(* CoDeSys 2.3.9.41 project: GermesLib_1_2.pro *)
(* Libraries: PID_Regulators.lib 6.11.19 15:29:27, Util.lib 18.5.10 15:14:28, STANDARD.LIB 4.10.05 11:14:46, IECSFC.LIB 13.4.06 15:51:28, ANALYZATION.LIB 5.10.99 09:05:06 *)

(* PLC configuration (modules and I/O channels)
Fast discrete inputs [I_SIMPLE_INPUT] node 0, in %IB0 out %QB0 {Filtrationtime = 10}
  DD1_DI0 AT %IX0.0 [BitInput] резерв
  DD1_DI1 AT %IX0.1 [BitInput] резерв
  DD1_DI2 AT %IX0.2 [BitInput] резерв
  DD1_DI3 AT %IX0.3 [BitInput] резерв
Discrete inputs [ID130] node 1, in %IB1 out %QB1 {Filtrationtime_GeneralINP = 10; Visibility = No; PinCount = 12}
  AT %IB1.0 [ByteInput] 8 discrete inputs
  AT %IB1.1 [ByteInput] 4 discrete inputs
Discrete outputs [ID131] node 2, in %IB2 out %QB2 {SafeValueByte = 0; SafeValueByteM = 0; Visibility = No; PinCount = 12}
  AT %QB2.0 [ByteOutput] 8 discrete outputs
  AT %QB2.1 [ByteOutput] 4 discrete outputs
Fast analog inputs [ID125] node 3, in %IB3 out %QB3 {Flt_Comm = 50Hz 2Por}
  DD1_AI0 AT %IR3.0 [FloatInputP] AI #1 - датчик температуры в помещении (метран) {AIN_TYPE = 4-20 mA; Peak_Filtr = 200; Flt_Ch = Off; TauRC = 10; MinFV = 0; MaxFV = 100}
  DD1_AI1 AT %IR3.1 [FloatInputP] AI #2 - расходомер FT01.01 (на входе, до отстойника) {AIN_TYPE = 4-20 mA; Peak_Filtr = 200; Flt_Ch = Off; TauRC = 10; MinFV = 0; MaxFV = 600}
  DD1_AI2 AT %IR3.2 [FloatInputP] AI #3 - расходомер FT01.02 (на выходе, после отстойника) {AIN_TYPE = 4-20 mA; Peak_Filtr = 200; Flt_Ch = Off; TauRC = 10; MinFV = 0; MaxFV = 600}
  DD1_AI3 AT %IR3.3 [FloatInputP] AI #4 - рН-метр QE01.01 (на входе, до отстойника) {AIN_TYPE = 4-20 mA; Peak_Filtr = 200; Flt_Ch = Off; TauRC = 10; MinFV = 0; MaxFV = 14}
  DD1_AI4 AT %IR3.4 [FloatInputP] AI #5 - рН-метр QE01.02 (на выходе, после отстойника) {AIN_TYPE = 4-20 mA; Peak_Filtr = 200; Flt_Ch = Off; TauRC = 10; MinFV = 0; MaxFV = 14}
  DD1_AI5 AT %IR3.5 [FloatInputP] AI #6 - сигнал от ФПК, давление на входе {AIN_TYPE = 4-20 mA; Peak_Filtr = 200; Flt_Ch = Off; TauRC = 10; MinFV = 0; MaxFV = 16}
  DD1_AI6 AT %IR3.6 [FloatInputP] AI #7 - резерв {AIN_TYPE = 4-20 mA; Peak_Filtr = 200; Flt_Ch = Off; TauRC = 10; MinFV = 0; MaxFV = 20000.0}
  DD1_AI7 AT %IR3.7 [FloatInputP] AI#8 - резерв {AIN_TYPE = 4-20 mA; Peak_Filtr = 200; Flt_Ch = Off; TauRC = 10; MinFV = 0; MaxFV = 20000.0}
  AT %IW3.8 [WordInput] AI read time (10ms)
Analog outputs [ID126] node 4, in %IB4 out %QB4
  DD1_AO0 AT %QR4.0 [FloatOutputP] AO #1 - управление ЧРП Н01.05 (поддержание расхода по расходомеру FT01.02) {AOUT_TYPE = 4-20 mA; SafeValueREAL = 0.0}
  DD1_AO1 AT %QR4.1 [FloatOutputP] AO #2 - управление ЧРП НД08.03/01 (подача флокулянта на входе, до отстойника, по FT01.01) {AOUT_TYPE = 4-20 mA; SafeValueREAL = 0.0}
  DD1_AO2 AT %QR4.2 [FloatOutputP] AO #3 - управление ЧРП НД08.03/02 (подача флокулянта на входе, до отстойника, по FT01.01) {AOUT_TYPE = 4-20 mA; SafeValueREAL = 0.0}
  DD1_AO3 AT %QR4.3 [FloatOutputP] AO #4 - управление НД05.02/01 (подача 10%NaCl из УПГ на входе, до отстойника, по FT01.01) {AOUT_TYPE = 4-20 mA; SafeValueREAL = 0.0}
Special input [ID103] node 5, in %IB5 out %QB5 {Filtrationtime = 1000; PinCount = 1; WatchDogPeriod = 400; PollPeriod = 3000; Visibility = No}
  AT %IX5.0 [BitInput] Special input
Special output [ID104] node 6, in %IB6 out %QB6 {Visibility = No; PinCount = 1}
  AT %QX6.0 [BitOutput] Special output
lastAddress AT %QD7.0 [DWordOutput] Last address
lastError AT %QW7.1 [WordOutput] Last error
RS-485-1 [COM1_USART] node 0, in %IB7.0 out %QB7.0 {CommunicationSpeed = 9600; Parity = EVEN; BitLength = 8 bits; StopLength = One stop bit; InterfaceType = RS485; FrameOriented = RTU; Timeout = 0; Visibility = No}
Universal Modbus device [ID2000] node 1, in %IB7.1 out %QB7.1 {ModuleIP = 10:0:0:102; ServiceTimeout = 20; TCPport = 502; NetMode = Serial; ModuleSlaveAddress = 2; RequestType = Both; PeriodOfService = 100; Visibility = No; RepeatCounter = 0; ByteSequence = Trace_mode}
  AT %QB7.1.0 [ComChannel] Command (0xff - Start)
DD2_DO AT %QD7.1.0.0 [DWordOutput] регистр 0, команда 0х0f
Universal Modbus device [ID2000] node 2, in %IB7.2 out %QB7.2 {ModuleIP = 10:0:0:103; ServiceTimeout = 20; TCPport = 502; NetMode = Serial; ModuleSlaveAddress = 3; RequestType = Both; PeriodOfService = 100; Visibility = No; RepeatCounter = 0; ByteSequence = Trace_mode}
  AT %QB7.2.0 [ComChannel] Command (0xff - Start)
DD3_DO AT %QD7.2.0.0 [DWordOutput]
Universal Modbus device [ID2000] node 3, in %IB7.3 out %QB7.3 {ModuleIP = 10:0:0:104; ServiceTimeout = 20; TCPport = 502; NetMode = Serial; ModuleSlaveAddress = 4; RequestType = Both; PeriodOfService = 100; Visibility = No; RepeatCounter = 0; ByteSequence = Trace_mode}
  AT %QB7.3.0 [ComChannel] Command (0xff - Start)
  32bit output module [ID2006] node 0, in %IB7.3.0 out %QB7.3.0 {ModbusAddress = 0; Command_write_regs = Force multiple coils (0x0f); Visibility = No}
    DD4_DO AT %QD7.3.0.0 [DWordOutput]
Universal Modbus device [ID2000] node 4, in %IB7.4 out %QB7.4 {ModuleIP = 10:0:0:105; ServiceTimeout = 20; TCPport = 502; NetMode = Serial; ModuleSlaveAddress = 5; RequestType = Both; PeriodOfService = 100; Visibility = No; RepeatCounter = 0; ByteSequence = Trace_mode}
  AT %QB7.4.0 [ComChannel] Command (0xff - Start)
DD5_DI AT %ID7.4.0.0 [DWordInput]
Universal Modbus device [ID2000] node 5, in %IB7.5 out %QB7.5 {ModuleIP = 10:0:0:106; ServiceTimeout = 20; TCPport = 502; NetMode = Serial; ModuleSlaveAddress = 6; RequestType = Both; PeriodOfService = 100; Visibility = No; RepeatCounter = 0; ByteSequence = Trace_mode}
  AT %QB7.5.0 [ComChannel] Command (0xff - Start)
DD6_DI AT %ID7.5.0.0 [DWordInput]
Universal Modbus device [ID2000] node 6, in %IB7.6 out %QB7.6 {ModuleIP = 10:0:0:107; ServiceTimeout = 20; TCPport = 502; NetMode = Serial; ModuleSlaveAddress = 7; RequestType = Both; PeriodOfService = 100; Visibility = No; RepeatCounter = 0; ByteSequence = Trace_mode}
  AT %QB7.6.0 [ComChannel] Command (0xff - Start)
DD7_DI AT %ID7.6.0.0 [DWordInput]
Universal Modbus device [ID2000] node 7, in %IB7.7 out %QB7.7 {ModuleIP = 10:0:0:108; ServiceTimeout = 20; TCPport = 502; NetMode = Serial; ModuleSlaveAddress = 8; RequestType = Both; PeriodOfService = 100; Visibility = No; RepeatCounter = 0; ByteSequence = Trace_mode}
  AT %QB7.7.0 [ComChannel] Command (0xff - Start)
DD8_DI AT %ID7.7.0.0 [DWordInput]
Universal Modbus device [ID2000] node 8, in %IB7.8 out %QB7.8 {ModuleIP = 10:0:0:109; ServiceTimeout = 20; TCPport = 502; NetMode = Serial; ModuleSlaveAddress = 9; RequestType = Both; PeriodOfService = 100; Visibility = No; RepeatCounter = 0; ByteSequence = Trace_mode}
  AT %QB7.8.0 [ComChannel] Command (0xff - Start)
DD9_DI AT %ID7.8.0.0 [DWordInput]
Universal Modbus device [ID2000] node 9, in %IB7.9 out %QB7.9 {ModuleIP = 10:0:0:110; ServiceTimeout = 20; TCPport = 502; NetMode = Serial; ModuleSlaveAddress = 10; RequestType = Both; PeriodOfService = 100; Visibility = No; RepeatCounter = 0; ByteSequence = Trace_mode}
  AT %QB7.9.0 [ComChannel] Command (0xff - Start)
DD10_AO0 AT %QW7.9.0.0 [WordOutput] управление 4...20мА НД05.02/02
DD10_AO1 AT %QW7.9.1.0 [WordOutput] управление 4...20мА НД06.02/01
DD10_AO2 AT %QW7.9.2.0 [WordOutput] управление 4...20мА НД06.02/02
DD10_AO3 AT %QW7.9.3.0 [WordOutput] управление 4...20мА НД06.03/01
DD10_AO4 AT %QW7.9.4.0 [WordOutput] управление 4...20мА НД06.03/02
DD10_AO5 AT %QW7.9.5.0 [WordOutput] управление 4...20мА НД07.03/01
DD10_AO6 AT %QW7.9.6.0 [WordOutput] управление 4...20мА НД07.03/02
DD10_AO7 AT %QW7.9.7.0 [WordOutput] управление 4...20мА НД08.04
Universal Modbus device [ID2000] node 10, in %IB7.10 out %QB7.10 {ModuleIP = 10:0:0:223; ServiceTimeout = 20; TCPport = 502; NetMode = Serial; ModuleSlaveAddress = 11; RequestType = By value change; PeriodOfService = 100; Visibility = No; RepeatCounter = 0; ByteSequence = Trace_mode}
  AT %QB7.10.0 [ComChannel] Command (0xff - Start)
AT %QB7.10.0.0 [ByteOutput]
Universal Modbus device [ID2000] node 11, in %IB7.11 out %QB7.11 {ModuleIP = 10:0:0:223; ServiceTimeout = 20; TCPport = 502; NetMode = Serial; ModuleSlaveAddress = 11; RequestType = By poll time; PeriodOfService = 100; Visibility = No; RepeatCounter = 0; ByteSequence = Trace_mode}
  AT %QB7.11.0 [ComChannel] Command (0xff - Start)
AT %IB7.11.0.0 [ByteInput]
Universal Modbus device [ID2000] node 12, in %IB7.12 out %QB7.12 {ModuleIP = 10:0:0:223; ServiceTimeout = 20; TCPport = 502; NetMode = Serial; ModuleSlaveAddress = 12; RequestType = By value change; PeriodOfService = 100; Visibility = No; RepeatCounter = 0; ByteSequence = Trace_mode}
  AT %QB7.12.0 [ComChannel] Command (0xff - Start)
AT %QB7.12.0.0 [ByteOutput]
Universal Modbus device [ID2000] node 13, in %IB7.13 out %QB7.13 {ModuleIP = 10:0:0:223; ServiceTimeout = 20; TCPport = 502; NetMode = Serial; ModuleSlaveAddress = 12; RequestType = By poll time; PeriodOfService = 100; Visibility = No; RepeatCounter = 0; ByteSequence = Trace_mode}
  AT %QB7.13.0 [ComChannel] Command (0xff - Start)
AT %IB7.13.0.0 [ByteInput]
AT %QD8.0 [DWordOutput] Last address
AT %QW8.1 [WordOutput] Last error
RS-232 [COM2_USART] node 0, in %IB8.0 out %QB8.0 {CommunicationSpeed = 57600; Parity = NO PARITY CHECK; BitLength = 8 bits; StopLength = One stop bit; InterfaceType = RS232; FrameOriented = RTU; Timeout = 0; Visibility = No}
AT %QB8.1.0 [ComChannel] Command (0xff - Start)
Real output module [ID2008] node 0, in %IB8.1.0 out %QB8.1.0 {ModbusAddress = 256; Command_write_regs = Preset multiple Registers (0x10); Visibility = No}
  panFT0101value AT %QD8.1.0.0 [FloatOutput]
Real output module [ID2008] node 1, in %IB8.1.1 out %QB8.1.1 {ModbusAddress = 258; Command_write_regs = Preset multiple Registers (0x10); Visibility = No}
  panQE0101value AT %QD8.1.1.0 [FloatOutput]
Real output module [ID2008] node 2, in %IB8.1.2 out %QB8.1.2 {ModbusAddress = 260; Command_write_regs = Preset multiple Registers (0x10); Visibility = No}
  panFT0102value AT %QD8.1.2.0 [FloatOutput]
Real output module [ID2008] node 3, in %IB8.1.3 out %QB8.1.3 {ModbusAddress = 262; Command_write_regs = Preset multiple Registers (0x10); Visibility = No}
  panQE0102value AT %QD8.1.3.0 [FloatOutput]
Real output module [ID2008] node 4, in %IB8.1.4 out %QB8.1.4 {ModbusAddress = 264; Command_write_regs = Preset multiple Registers (0x10); Visibility = No}
  panFPKpressureValue AT %QD8.1.4.0 [FloatOutput]
Real output module [ID2008] node 5, in %IB8.1.5 out %QB8.1.5 {ModbusAddress = 266; Command_write_regs = Preset multiple Registers (0x10); Visibility = No}
  panFQS0301total AT %QD8.1.5.0 [FloatOutput]
Real output module [ID2008] node 6, in %IB8.1.6 out %QB8.1.6 {ModbusAddress = 268; Command_write_regs = Preset multiple Registers (0x10); Visibility = No}
  panTemperature AT %QD8.1.6.0 [FloatOutput]
Register output module [ID2004] node 7, in %IB8.1.7 out %QB8.1.7 {ModbusAddress = 270; Command_write_one_reg = Write multiple registers(0x10); Visibility = No}
  panND050201workDays AT %QW8.1.7.0 [WordOutput]
Register output module [ID2004] node 8, in %IB8.1.8 out %QB8.1.8 {ModbusAddress = 271; Command_write_one_reg = Write multiple registers(0x10); Visibility = No}
  panND050201workHours AT %QW8.1.8.0 [WordOutput]
Register output module [ID2004] node 9, in %IB8.1.9 out %QB8.1.9 {ModbusAddress = 272; Command_write_one_reg = Write multiple registers(0x10); Visibility = No}
  panND050201workMinutes AT %QW8.1.9.0 [WordOutput]
Register output module [ID2004] node 10, in %IB8.1.10 out %QB8.1.10 {ModbusAddress = 273; Command_write_one_reg = Write multiple registers(0x10); Visibility = No}
  panND050201workSeconds AT %QW8.1.10.0 [WordOutput]
Register output module [ID2004] node 11, in %IB8.1.11 out %QB8.1.11 {ModbusAddress = 274; Command_write_one_reg = Write multiple registers(0x10); Visibility = No}
  panND050202workDays AT %QW8.1.11.0 [WordOutput]
Register output module [ID2004] node 12, in %IB8.1.12 out %QB8.1.12 {ModbusAddress = 275; Command_write_one_reg = Write multiple registers(0x10); Visibility = No}
  panND050202workHours AT %QW8.1.12.0 [WordOutput]
Register output module [ID2004] node 13, in %IB8.1.13 out %QB8.1.13 {ModbusAddress = 276; Command_write_one_reg = Write multiple registers(0x10); Visibility = No}
  panND050202workMinutes AT %QW8.1.13.0 [WordOutput]
Register output module [ID2004] node 14, in %IB8.1.14 out %QB8.1.14 {ModbusAddress = 277; Command_write_one_reg = Write multiple registers(0x10); Visibility = No}
  panND050202workSeconds AT %QW8.1.14.0 [WordOutput]
Register output module [ID2004] node 15, in %IB8.1.15 out %QB8.1.15 {ModbusAddress = 278; Command_write_one_reg = Write multiple registers(0x10); Visibility = No}
  panND0502counterP1 AT %QW8.1.15.0 [WordOutput]
Register output module [ID2004] node 16, in %IB8.1.16 out %QB8.1.16 {ModbusAddress = 279; Command_write_one_reg = Write multiple registers(0x10); Visibility = No}
  panND0502counterP2 AT %QW8.1.16.0 [WordOutput]
Register output module [ID2004] node 17, in %IB8.1.17 out %QB8.1.17 {ModbusAddress = 280; Command_write_one_reg = Write multiple registers(0x10); Visibility = No}
  panND060201workDays AT %QW8.1.17.0 [WordOutput]
Register output module [ID2004] node 18, in %IB8.1.18 out %QB8.1.18 {ModbusAddress = 281; Command_write_one_reg = Write multiple registers(0x10); Visibility = No}
  panND060201workHours AT %QW8.1.18.0 [WordOutput]
Register output module [ID2004] node 19, in %IB8.1.19 out %QB8.1.19 {ModbusAddress = 282; Command_write_one_reg = Write multiple registers(0x10); Visibility = No}
  panND060201workMinutes AT %QW8.1.19.0 [WordOutput]
Register output module [ID2004] node 20, in %IB8.1.20 out %QB8.1.20 {ModbusAddress = 283; Command_write_one_reg = Write multiple registers(0x10); Visibility = No}
  panND060201workSeconds AT %QW8.1.20.0 [WordOutput]
Register output module [ID2004] node 21, in %IB8.1.21 out %QB8.1.21 {ModbusAddress = 284; Command_write_one_reg = Write multiple registers(0x10); Visibility = No}
  panND060202workDays AT %QW8.1.21.0 [WordOutput]
Register output module [ID2004] node 22, in %IB8.1.22 out %QB8.1.22 {ModbusAddress = 285; Command_write_one_reg = Write multiple registers(0x10); Visibility = No}
  panND060202workHours AT %QW8.1.22.0 [WordOutput]
Register output module [ID2004] node 23, in %IB8.1.23 out %QB8.1.23 {ModbusAddress = 286; Command_write_one_reg = Write multiple registers(0x10); Visibility = No}
  panND060202workMinutes AT %QW8.1.23.0 [WordOutput]
Register output module [ID2004] node 24, in %IB8.1.24 out %QB8.1.24 {ModbusAddress = 287; Command_write_one_reg = Write multiple registers(0x10); Visibility = No}
  panND060202workSeconds AT %QW8.1.24.0 [WordOutput]
Register output module [ID2004] node 25, in %IB8.1.25 out %QB8.1.25 {ModbusAddress = 288; Command_write_one_reg = Write multiple registers(0x10); Visibility = No}
  panND0602counterP1 AT %QW8.1.25.0 [WordOutput]
Register output module [ID2004] node 26, in %IB8.1.26 out %QB8.1.26 {ModbusAddress = 289; Command_write_one_reg = Write multiple registers(0x10); Visibility = No}
  panND0602counterP2 AT %QW8.1.26.0 [WordOutput]
Register output module [ID2004] node 27, in %IB8.1.27 out %QB8.1.27 {ModbusAddress = 290; Command_write_one_reg = Write multiple registers(0x10); Visibility = No}
  panND060301workDays AT %QW8.1.27.0 [WordOutput]
Register output module [ID2004] node 28, in %IB8.1.28 out %QB8.1.28 {ModbusAddress = 291; Command_write_one_reg = Write multiple registers(0x10); Visibility = No}
  panND060301workHours AT %QW8.1.28.0 [WordOutput]
Register output module [ID2004] node 29, in %IB8.1.29 out %QB8.1.29 {ModbusAddress = 292; Command_write_one_reg = Write multiple registers(0x10); Visibility = No}
  panND060301workMinutes AT %QW8.1.29.0 [WordOutput]
Register output module [ID2004] node 30, in %IB8.1.30 out %QB8.1.30 {ModbusAddress = 293; Command_write_one_reg = Write multiple registers(0x10); Visibility = No}
  panND060301workSeconds AT %QW8.1.30.0 [WordOutput]
Register output module [ID2004] node 31, in %IB8.1.31 out %QB8.1.31 {ModbusAddress = 294; Command_write_one_reg = Write multiple registers(0x10); Visibility = No}
  panND060302workDays AT %QW8.1.31.0 [WordOutput]
Register output module [ID2004] node 32, in %IB8.1.32 out %QB8.1.32 {ModbusAddress = 295; Command_write_one_reg = Write multiple registers(0x10); Visibility = No}
  panND060302workHours AT %QW8.1.32.0 [WordOutput]
Register output module [ID2004] node 33, in %IB8.1.33 out %QB8.1.33 {ModbusAddress = 296; Command_write_one_reg = Write multiple registers(0x10); Visibility = No}
  panND060302workMinutes AT %QW8.1.33.0 [WordOutput]
Register output module [ID2004] node 34, in %IB8.1.34 out %QB8.1.34 {ModbusAddress = 297; Command_write_one_reg = Write multiple registers(0x10); Visibility = No}
  panND060302workSeconds AT %QW8.1.34.0 [WordOutput]
Register output module [ID2004] node 35, in %IB8.1.35 out %QB8.1.35 {ModbusAddress = 298; Command_write_one_reg = Write multiple registers(0x10); Visibility = No}
  panND0603counterP1 AT %QW8.1.35.0 [WordOutput]
Register output module [ID2004] node 36, in %IB8.1.36 out %QB8.1.36 {ModbusAddress = 299; Command_write_one_reg = Write multiple registers(0x10); Visibility = No}
  panND0603counterP2 AT %QW8.1.36.0 [WordOutput]
Register output module [ID2004] node 37, in %IB8.1.37 out %QB8.1.37 {ModbusAddress = 300; Command_write_one_reg = Write multiple registers(0x10); Visibility = No}
  panND070301workDays AT %QW8.1.37.0 [WordOutput]
Register output module [ID2004] node 38, in %IB8.1.38 out %QB8.1.38 {ModbusAddress = 301; Command_write_one_reg = Write multiple registers(0x10); Visibility = No}
  panND070301workHours AT %QW8.1.38.0 [WordOutput]
Register output module [ID2004] node 39, in %IB8.1.39 out %QB8.1.39 {ModbusAddress = 302; Command_write_one_reg = Write multiple registers(0x10); Visibility = No}
  panND070301workMinutes AT %QW8.1.39.0 [WordOutput]
Register output module [ID2004] node 40, in %IB8.1.40 out %QB8.1.40 {ModbusAddress = 303; Command_write_one_reg = Write multiple registers(0x10); Visibility = No}
  panND070301workSeconds AT %QW8.1.40.0 [WordOutput]
Register output module [ID2004] node 41, in %IB8.1.41 out %QB8.1.41 {ModbusAddress = 304; Command_write_one_reg = Write multiple registers(0x10); Visibility = No}
  panND070302workDays AT %QW8.1.41.0 [WordOutput]
Register output module [ID2004] node 42, in %IB8.1.42 out %QB8.1.42 {ModbusAddress = 305; Command_write_one_reg = Write multiple registers(0x10); Visibility = No}
  panND070302workHours AT %QW8.1.42.0 [WordOutput]
Register output module [ID2004] node 43, in %IB8.1.43 out %QB8.1.43 {ModbusAddress = 306; Command_write_one_reg = Write multiple registers(0x10); Visibility = No}
  panND070302workMinutes AT %QW8.1.43.0 [WordOutput]
Register output module [ID2004] node 44, in %IB8.1.44 out %QB8.1.44 {ModbusAddress = 307; Command_write_one_reg = Write multiple registers(0x10); Visibility = No}
  panND070302workSeconds AT %QW8.1.44.0 [WordOutput]
Register output module [ID2004] node 45, in %IB8.1.45 out %QB8.1.45 {ModbusAddress = 308; Command_write_one_reg = Write multiple registers(0x10); Visibility = No}
  panND0703counterP1 AT %QW8.1.45.0 [WordOutput]
Register output module [ID2004] node 46, in %IB8.1.46 out %QB8.1.46 {ModbusAddress = 309; Command_write_one_reg = Write multiple registers(0x10); Visibility = No}
  panND0703counterP2 AT %QW8.1.46.0 [WordOutput]
Register output module [ID2004] node 47, in %IB8.1.47 out %QB8.1.47 {ModbusAddress = 310; Command_write_one_reg = Write multiple registers(0x10); Visibility = No}
  panND080301workDays AT %QW8.1.47.0 [WordOutput]
Register output module [ID2004] node 48, in %IB8.1.48 out %QB8.1.48 {ModbusAddress = 311; Command_write_one_reg = Write multiple registers(0x10); Visibility = No}
  panND080301workHours AT %QW8.1.48.0 [WordOutput]
Register output module [ID2004] node 49, in %IB8.1.49 out %QB8.1.49 {ModbusAddress = 312; Command_write_one_reg = Write multiple registers(0x10); Visibility = No}
  panND080301workMinutes AT %QW8.1.49.0 [WordOutput]
Register output module [ID2004] node 50, in %IB8.1.50 out %QB8.1.50 {ModbusAddress = 313; Command_write_one_reg = Write multiple registers(0x10); Visibility = No}
  panND080301workSeconds AT %QW8.1.50.0 [WordOutput]
Register output module [ID2004] node 51, in %IB8.1.51 out %QB8.1.51 {ModbusAddress = 314; Command_write_one_reg = Write multiple registers(0x10); Visibility = No}
  panND080302workDays AT %QW8.1.51.0 [WordOutput]
Register output module [ID2004] node 52, in %IB8.1.52 out %QB8.1.52 {ModbusAddress = 315; Command_write_one_reg = Write multiple registers(0x10); Visibility = No}
  panND080302workHours AT %QW8.1.52.0 [WordOutput]
Register output module [ID2004] node 53, in %IB8.1.53 out %QB8.1.53 {ModbusAddress = 316; Command_write_one_reg = Write multiple registers(0x10); Visibility = No}
  panND080302workMinutes AT %QW8.1.53.0 [WordOutput]
Register output module [ID2004] node 54, in %IB8.1.54 out %QB8.1.54 {ModbusAddress = 317; Command_write_one_reg = Write multiple registers(0x10); Visibility = No}
  panND080302workSeconds AT %QW8.1.54.0 [WordOutput]
Register output module [ID2004] node 55, in %IB8.1.55 out %QB8.1.55 {ModbusAddress = 318; Command_write_one_reg = Write multiple registers(0x10); Visibility = No}
  panND0803counterP1 AT %QW8.1.55.0 [WordOutput]
Register output module [ID2004] node 56, in %IB8.1.56 out %QB8.1.56 {ModbusAddress = 319; Command_write_one_reg = Write multiple registers(0x10); Visibility = No}
  panND0803counterP2 AT %QW8.1.56.0 [WordOutput]
Register output module [ID2004] node 57, in %IB8.1.57 out %QB8.1.57 {ModbusAddress = 320; Command_write_one_reg = Write multiple registers(0x10); Visibility = No}
  panN010501workDays AT %QW8.1.57.0 [WordOutput]
Register output module [ID2004] node 58, in %IB8.1.58 out %QB8.1.58 {ModbusAddress = 321; Command_write_one_reg = Write multiple registers(0x10); Visibility = No}
  panN010501workHours AT %QW8.1.58.0 [WordOutput]
Register output module [ID2004] node 59, in %IB8.1.59 out %QB8.1.59 {ModbusAddress = 322; Command_write_one_reg = Write multiple registers(0x10); Visibility = No}
  panN010501workMinutes AT %QW8.1.59.0 [WordOutput]
Register output module [ID2004] node 60, in %IB8.1.60 out %QB8.1.60 {ModbusAddress = 323; Command_write_one_reg = Write multiple registers(0x10); Visibility = No}
  panN010501workSeconds AT %QW8.1.60.0 [WordOutput]
Register output module [ID2004] node 61, in %IB8.1.61 out %QB8.1.61 {ModbusAddress = 324; Command_write_one_reg = Write multiple registers(0x10); Visibility = No}
  panN010502workDays AT %QW8.1.61.0 [WordOutput]
Register output module [ID2004] node 62, in %IB8.1.62 out %QB8.1.62 {ModbusAddress = 325; Command_write_one_reg = Write multiple registers(0x10); Visibility = No}
  panN010502workHours AT %QW8.1.62.0 [WordOutput]
Register output module [ID2004] node 63, in %IB8.1.63 out %QB8.1.63 {ModbusAddress = 326; Command_write_one_reg = Write multiple registers(0x10); Visibility = No}
  panN010502workMinutes AT %QW8.1.63.0 [WordOutput]
Register output module [ID2004] node 64, in %IB8.1.64 out %QB8.1.64 {ModbusAddress = 327; Command_write_one_reg = Write multiple registers(0x10); Visibility = No}
  panN010502workSeconds AT %QW8.1.64.0 [WordOutput]
Register output module [ID2004] node 65, in %IB8.1.65 out %QB8.1.65 {ModbusAddress = 328; Command_write_one_reg = Write multiple registers(0x10); Visibility = No}
  panN0105counterP1 AT %QW8.1.65.0 [WordOutput]
Register output module [ID2004] node 66, in %IB8.1.66 out %QB8.1.66 {ModbusAddress = 329; Command_write_one_reg = Write multiple registers(0x10); Visibility = No}
  panN0105counterP2 AT %QW8.1.66.0 [WordOutput]
Register output module [ID2004] node 67, in %IB8.1.67 out %QB8.1.67 {ModbusAddress = 330; Command_write_one_reg = Write multiple registers(0x10); Visibility = No}
  panN020401workDays AT %QW8.1.67.0 [WordOutput]
Register output module [ID2004] node 68, in %IB8.1.68 out %QB8.1.68 {ModbusAddress = 331; Command_write_one_reg = Write multiple registers(0x10); Visibility = No}
  panN020401workHours AT %QW8.1.68.0 [WordOutput]
Register output module [ID2004] node 69, in %IB8.1.69 out %QB8.1.69 {ModbusAddress = 332; Command_write_one_reg = Write multiple registers(0x10); Visibility = No}
  panN020401workMinutes AT %QW8.1.69.0 [WordOutput]
Register output module [ID2004] node 70, in %IB8.1.70 out %QB8.1.70 {ModbusAddress = 333; Command_write_one_reg = Write multiple registers(0x10); Visibility = No}
  panN020401workSeconds AT %QW8.1.70.0 [WordOutput]
Register output module [ID2004] node 71, in %IB8.1.71 out %QB8.1.71 {ModbusAddress = 334; Command_write_one_reg = Write multiple registers(0x10); Visibility = No}
  panN020402workDays AT %QW8.1.71.0 [WordOutput]
Register output module [ID2004] node 72, in %IB8.1.72 out %QB8.1.72 {ModbusAddress = 335; Command_write_one_reg = Write multiple registers(0x10); Visibility = No}
  panN020402workHours AT %QW8.1.72.0 [WordOutput]
Register output module [ID2004] node 73, in %IB8.1.73 out %QB8.1.73 {ModbusAddress = 336; Command_write_one_reg = Write multiple registers(0x10); Visibility = No}
  panN020402workMinutes AT %QW8.1.73.0 [WordOutput]
Register output module [ID2004] node 74, in %IB8.1.74 out %QB8.1.74 {ModbusAddress = 337; Command_write_one_reg = Write multiple registers(0x10); Visibility = No}
  panN020402workSeconds AT %QW8.1.74.0 [WordOutput]
Register output module [ID2004] node 75, in %IB8.1.75 out %QB8.1.75 {ModbusAddress = 338; Command_write_one_reg = Write multiple registers(0x10); Visibility = No}
  panN0204counterP1 AT %QW8.1.75.0 [WordOutput]
Register output module [ID2004] node 76, in %IB8.1.76 out %QB8.1.76 {ModbusAddress = 339; Command_write_one_reg = Write multiple registers(0x10); Visibility = No}
  panN0204counterP2 AT %QW8.1.76.0 [WordOutput]
Register output module [ID2004] node 77, in %IB8.1.77 out %QB8.1.77 {ModbusAddress = 340; Command_write_one_reg = Write multiple registers(0x10); Visibility = No}
  panN040401workDays AT %QW8.1.77.0 [WordOutput]
Register output module [ID2004] node 78, in %IB8.1.78 out %QB8.1.78 {ModbusAddress = 341; Command_write_one_reg = Write multiple registers(0x10); Visibility = No}
  panN040401workHours AT %QW8.1.78.0 [WordOutput]
Register output module [ID2004] node 79, in %IB8.1.79 out %QB8.1.79 {ModbusAddress = 342; Command_write_one_reg = Write multiple registers(0x10); Visibility = No}
  panN040401workMinutes AT %QW8.1.79.0 [WordOutput]
Register output module [ID2004] node 80, in %IB8.1.80 out %QB8.1.80 {ModbusAddress = 343; Command_write_one_reg = Write multiple registers(0x10); Visibility = No}
  panN040401workSeconds AT %QW8.1.80.0 [WordOutput]
Register output module [ID2004] node 81, in %IB8.1.81 out %QB8.1.81 {ModbusAddress = 344; Command_write_one_reg = Write multiple registers(0x10); Visibility = No}
  panN040402workDays AT %QW8.1.81.0 [WordOutput]
Register output module [ID2004] node 82, in %IB8.1.82 out %QB8.1.82 {ModbusAddress = 345; Command_write_one_reg = Write multiple registers(0x10); Visibility = No}
  panN040402workHours AT %QW8.1.82.0 [WordOutput]
Register output module [ID2004] node 83, in %IB8.1.83 out %QB8.1.83 {ModbusAddress = 346; Command_write_one_reg = Write multiple registers(0x10); Visibility = No}
  panN040402workMinutes AT %QW8.1.83.0 [WordOutput]
Register output module [ID2004] node 84, in %IB8.1.84 out %QB8.1.84 {ModbusAddress = 347; Command_write_one_reg = Write multiple registers(0x10); Visibility = No}
  panN040402workSeconds AT %QW8.1.84.0 [WordOutput]
Register output module [ID2004] node 85, in %IB8.1.85 out %QB8.1.85 {ModbusAddress = 348; Command_write_one_reg = Write multiple registers(0x10); Visibility = No}
  panN0404counterP1 AT %QW8.1.85.0 [WordOutput]
Register output module [ID2004] node 86, in %IB8.1.86 out %QB8.1.86 {ModbusAddress = 349; Command_write_one_reg = Write multiple registers(0x10); Visibility = No}
  panN0404counterP2 AT %QW8.1.86.0 [WordOutput]
Register output module [ID2004] node 87, in %IB8.1.87 out %QB8.1.87 {ModbusAddress = 350; Command_write_one_reg = Write multiple registers(0x10); Visibility = No}
  panUFO030101workDays AT %QW8.1.87.0 [WordOutput]
Register output module [ID2004] node 88, in %IB8.1.88 out %QB8.1.88 {ModbusAddress = 351; Command_write_one_reg = Write multiple registers(0x10); Visibility = No}
  panUFO030101workHours AT %QW8.1.88.0 [WordOutput]
Register output module [ID2004] node 89, in %IB8.1.89 out %QB8.1.89 {ModbusAddress = 352; Command_write_one_reg = Write multiple registers(0x10); Visibility = No}
  panUFO030101workMinutes AT %QW8.1.89.0 [WordOutput]
Register output module [ID2004] node 90, in %IB8.1.90 out %QB8.1.90 {ModbusAddress = 353; Command_write_one_reg = Write multiple registers(0x10); Visibility = No}
  panUFO030101workSeconds AT %QW8.1.90.0 [WordOutput]
Register output module [ID2004] node 91, in %IB8.1.91 out %QB8.1.91 {ModbusAddress = 354; Command_write_one_reg = Write multiple registers(0x10); Visibility = No}
  panUFO030102workDays AT %QW8.1.91.0 [WordOutput]
Register output module [ID2004] node 92, in %IB8.1.92 out %QB8.1.92 {ModbusAddress = 355; Command_write_one_reg = Write multiple registers(0x10); Visibility = No}
  panUFO030102workHours AT %QW8.1.92.0 [WordOutput]
Register output module [ID2004] node 93, in %IB8.1.93 out %QB8.1.93 {ModbusAddress = 356; Command_write_one_reg = Write multiple registers(0x10); Visibility = No}
  panUFO030102workMinutes AT %QW8.1.93.0 [WordOutput]
Register output module [ID2004] node 94, in %IB8.1.94 out %QB8.1.94 {ModbusAddress = 357; Command_write_one_reg = Write multiple registers(0x10); Visibility = No}
  panUFO030102workSeconds AT %QW8.1.94.0 [WordOutput]
Register output module [ID2004] node 95, in %IB8.1.95 out %QB8.1.95 {ModbusAddress = 358; Command_write_one_reg = Write multiple registers(0x10); Visibility = No}
  panUFO0301counterP1 AT %QW8.1.95.0 [WordOutput]
Register output module [ID2004] node 96, in %IB8.1.96 out %QB8.1.96 {ModbusAddress = 359; Command_write_one_reg = Write multiple registers(0x10); Visibility = No}
  panUFO0301counterP2 AT %QW8.1.96.0 [WordOutput]
panVolumeToRegen AT %QD8.1.97.0 [FloatOutput]
8 bit output module [ID2002] node 98, in %IB8.1.98 out %QB8.1.98 {ModbusAddress = 256; Command_write_byte = Force multiply coils (0x0f); Visibility = No}
  AT %QB8.1.98.0 [ByteOutput]
8 bit output module [ID2002] node 99, in %IB8.1.99 out %QB8.1.99 {ModbusAddress = 264; Command_write_byte = Force multiply coils (0x0f); Visibility = No}
  AT %QB8.1.99.0 [ByteOutput]
8 bit output module [ID2002] node 100, in %IB8.1.100 out %QB8.1.100 {ModbusAddress = 272; Command_write_byte = Force multiply coils (0x0f); Visibility = No}
  AT %QB8.1.100.0 [ByteOutput]
8 bit output module [ID2002] node 101, in %IB8.1.101 out %QB8.1.101 {ModbusAddress = 280; Command_write_byte = Force multiply coils (0x0f); Visibility = No}
  AT %QB8.1.101.0 [ByteOutput]
8 bit output module [ID2002] node 102, in %IB8.1.102 out %QB8.1.102 {ModbusAddress = 288; Command_write_byte = Force multiply coils (0x0f); Visibility = No}
  AT %QB8.1.102.0 [ByteOutput]
8 bit output module [ID2002] node 103, in %IB8.1.103 out %QB8.1.103 {ModbusAddress = 296; Command_write_byte = Force multiply coils (0x0f); Visibility = No}
  AT %QB8.1.103.0 [ByteOutput]
8 bit output module [ID2002] node 104, in %IB8.1.104 out %QB8.1.104 {ModbusAddress = 304; Command_write_byte = Force multiply coils (0x0f); Visibility = No}
  AT %QB8.1.104.0 [ByteOutput]
8 bit output module [ID2002] node 105, in %IB8.1.105 out %QB8.1.105 {ModbusAddress = 312; Command_write_byte = Force multiply coils (0x0f); Visibility = No}
  AT %QB8.1.105.0 [ByteOutput]
8 bit output module [ID2002] node 106, in %IB8.1.106 out %QB8.1.106 {ModbusAddress = 320; Command_write_byte = Force multiply coils (0x0f); Visibility = No}
  AT %QB8.1.106.0 [ByteOutput]
8 bit output module [ID2002] node 107, in %IB8.1.107 out %QB8.1.107 {ModbusAddress = 328; Command_write_byte = Force multiply coils (0x0f); Visibility = No}
  AT %QB8.1.107.0 [ByteOutput]
8 bit output module [ID2002] node 108, in %IB8.1.108 out %QB8.1.108 {ModbusAddress = 336; Command_write_byte = Force multiply coils (0x0f); Visibility = No}
  AT %QB8.1.108.0 [ByteOutput]
8 bit output module [ID2002] node 109, in %IB8.1.109 out %QB8.1.109 {ModbusAddress = 344; Command_write_byte = Force multiply coils (0x0f); Visibility = No}
  AT %QB8.1.109.0 [ByteOutput]
8 bit output module [ID2002] node 110, in %IB8.1.110 out %QB8.1.110 {ModbusAddress = 352; Command_write_byte = Force multiply coils (0x0f); Visibility = No}
  AT %QB8.1.110.0 [ByteOutput]
8 bit output module [ID2002] node 111, in %IB8.1.111 out %QB8.1.111 {ModbusAddress = 360; Command_write_byte = Force multiply coils (0x0f); Visibility = No}
  AT %QB8.1.111.0 [ByteOutput]
8 bit output module [ID2002] node 112, in %IB8.1.112 out %QB8.1.112 {ModbusAddress = 368; Command_write_byte = Force multiply coils (0x0f); Visibility = No}
  AT %QB8.1.112.0 [ByteOutput]
8 bit output module [ID2002] node 113, in %IB8.1.113 out %QB8.1.113 {ModbusAddress = 376; Command_write_byte = Force multiply coils (0x0f); Visibility = No}
  AT %QB8.1.113.0 [ByteOutput]
8 bit output module [ID2002] node 114, in %IB8.1.114 out %QB8.1.114 {ModbusAddress = 384; Command_write_byte = Force multiply coils (0x0f); Visibility = No}
  AT %QB8.1.114.0 [ByteOutput]
8 bit output module [ID2002] node 115, in %IB8.1.115 out %QB8.1.115 {ModbusAddress = 392; Command_write_byte = Force multiply coils (0x0f); Visibility = No}
  AT %QB8.1.115.0 [ByteOutput]
8 bit output module [ID2002] node 116, in %IB8.1.116 out %QB8.1.116 {ModbusAddress = 400; Command_write_byte = Force multiply coils (0x0f); Visibility = No}
  AT %QB8.1.116.0 [ByteOutput]
8 bit output module [ID2002] node 117, in %IB8.1.117 out %QB8.1.117 {ModbusAddress = 408; Command_write_byte = Force multiply coils (0x0f); Visibility = No}
  AT %QB8.1.117.0 [ByteOutput]
8 bit output module [ID2002] node 118, in %IB8.1.118 out %QB8.1.118 {ModbusAddress = 416; Command_write_byte = Force multiply coils (0x0f); Visibility = No}
  AT %QB8.1.118.0 [ByteOutput]
8 bit output module [ID2002] node 119, in %IB8.1.119 out %QB8.1.119 {ModbusAddress = 424; Command_write_byte = Force multiply coils (0x0f); Visibility = No}
  AT %QB8.1.119.0 [ByteOutput]
8 bit output module [ID2002] node 120, in %IB8.1.120 out %QB8.1.120 {ModbusAddress = 432; Command_write_byte = Force multiply coils (0x0f); Visibility = No}
  AT %QB8.1.120.0 [ByteOutput]
8 bit output module [ID2002] node 121, in %IB8.1.121 out %QB8.1.121 {ModbusAddress = 440; Command_write_byte = Force multiply coils (0x0f); Visibility = No}
  AT %QB8.1.121.0 [ByteOutput]
8 bit output module [ID2002] node 122, in %IB8.1.122 out %QB8.1.122 {ModbusAddress = 448; Command_write_byte = Force multiply coils (0x0f); Visibility = No}
  AT %QB8.1.122.0 [ByteOutput]
8 bit output module [ID2002] node 123, in %IB8.1.123 out %QB8.1.123 {ModbusAddress = 456; Command_write_byte = Force multiply coils (0x0f); Visibility = No}
  AT %QB8.1.123.0 [ByteOutput]
8 bit output module [ID2002] node 124, in %IB8.1.124 out %QB8.1.124 {ModbusAddress = 464; Command_write_byte = Force multiply coils (0x0f); Visibility = No}
  AT %QB8.1.124.0 [ByteOutput]
8 bit output module [ID2002] node 125, in %IB8.1.125 out %QB8.1.125 {ModbusAddress = 472; Command_write_byte = Force multiply coils (0x0f); Visibility = No}
  AT %QB8.1.125.0 [ByteOutput]
8 bit output module [ID2002] node 126, in %IB8.1.126 out %QB8.1.126 {ModbusAddress = 480; Command_write_byte = Force multiply coils (0x0f); Visibility = No}
  AT %QB8.1.126.0 [ByteOutput]
8 bit output module [ID2002] node 127, in %IB8.1.127 out %QB8.1.127 {ModbusAddress = 488; Command_write_byte = Force multiply coils (0x0f); Visibility = No}
  AT %QB8.1.127.0 [ByteOutput]
8 bit output module [ID2002] node 128, in %IB8.1.128 out %QB8.1.128 {ModbusAddress = 496; Command_write_byte = Force multiply coils (0x0f); Visibility = No}
  AT %QB8.1.128.0 [ByteOutput]
8 bit output module [ID2002] node 129, in %IB8.1.129 out %QB8.1.129 {ModbusAddress = 504; Command_write_byte = Force multiply coils (0x0f); Visibility = No}
  AT %QB8.1.129.0 [ByteOutput]
8 bit output module [ID2002] node 130, in %IB8.1.130 out %QB8.1.130 {ModbusAddress = 512; Command_write_byte = Force multiply coils (0x0f); Visibility = No}
  AT %QB8.1.130.0 [ByteOutput]
8 bit output module [ID2002] node 131, in %IB8.1.131 out %QB8.1.131 {ModbusAddress = 520; Command_write_byte = Force multiply coils (0x0f); Visibility = No}
  AT %QB8.1.131.0 [ByteOutput]
8 bit output module [ID2002] node 132, in %IB8.1.132 out %QB8.1.132 {ModbusAddress = 528; Command_write_byte = Force multiply coils (0x0f); Visibility = No}
  AT %QB8.1.132.0 [ByteOutput]
8 bit output module [ID2002] node 133, in %IB8.1.133 out %QB8.1.133 {ModbusAddress = 632; Command_write_byte = Force multiply coils (0x0f); Visibility = No}
  AT %QB8.1.133.0 [ByteOutput]
  AT %QB8.1.134.0 [ByteOutput]
Universal Modbus device [ID2000] node 2, in %IB8.2 out %QB8.2 {ModuleIP = 10:0:0:223; ServiceTimeout = 150; TCPport = 502; NetMode = Serial; ModuleSlaveAddress = 1; RequestType = By poll time; PeriodOfService = 10; Visibility = No; RepeatCounter = 0; ByteSequence = Native}
  AT %QB8.2.0 [ComChannel] Command (0xff - Start)
  8 bit input module [ID2001] node 0, in %IB8.2.0 out %QB8.2.0 {ModbusAddress = 536; Command_read_byte = Read coils status (0x01); Visibility = No}
    AT %IB8.2.0.0 [ByteInput]
  8 bit input module [ID2001] node 1, in %IB8.2.1 out %QB8.2.1 {ModbusAddress = 544; Command_read_byte = Read coils status (0x01); Visibility = No}
    AT %IB8.2.1.0 [ByteInput]
  8 bit input module [ID2001] node 2, in %IB8.2.2 out %QB8.2.2 {ModbusAddress = 552; Command_read_byte = Read coils status (0x01); Visibility = No}
    AT %IB8.2.2.0 [ByteInput]
  8 bit input module [ID2001] node 3, in %IB8.2.3 out %QB8.2.3 {ModbusAddress = 560; Command_read_byte = Read coils status (0x01); Visibility = No}
    AT %IB8.2.3.0 [ByteInput]
  8 bit input module [ID2001] node 4, in %IB8.2.4 out %QB8.2.4 {ModbusAddress = 568; Command_read_byte = Read coils status (0x01); Visibility = No}
    AT %IB8.2.4.0 [ByteInput]
  8 bit input module [ID2001] node 5, in %IB8.2.5 out %QB8.2.5 {ModbusAddress = 576; Command_read_byte = Read coils status (0x01); Visibility = No}
    AT %IB8.2.5.0 [ByteInput]
  8 bit input module [ID2001] node 6, in %IB8.2.6 out %QB8.2.6 {ModbusAddress = 584; Command_read_byte = Read coils status (0x01); Visibility = No}
    AT %IB8.2.6.0 [ByteInput]
  8 bit input module [ID2001] node 7, in %IB8.2.7 out %QB8.2.7 {ModbusAddress = 592; Command_read_byte = Read coils status (0x01); Visibility = No}
    AT %IB8.2.7.0 [ByteInput]
  8 bit input module [ID2001] node 8, in %IB8.2.8 out %QB8.2.8 {ModbusAddress = 600; Command_read_byte = Read coils status (0x01); Visibility = No}
    AT %IB8.2.8.0 [ByteInput]
  8 bit input module [ID2001] node 9, in %IB8.2.9 out %QB8.2.9 {ModbusAddress = 608; Command_read_byte = Read coils status (0x01); Visibility = No}
    AT %IB8.2.9.0 [ByteInput]
  8 bit input module [ID2001] node 10, in %IB8.2.10 out %QB8.2.10 {ModbusAddress = 616; Command_read_byte = Read coils status (0x01); Visibility = No}
    AT %IB8.2.10.0 [ByteInput]
  8 bit input module [ID2001] node 11, in %IB8.2.11 out %QB8.2.11 {ModbusAddress = 624; Command_read_byte = Read coils status (0x01); Visibility = No}
    AT %IB8.2.11.0 [ByteInput]
  Real input module [ID2007] node 12, in %IB8.2.12 out %QB8.2.12 {ModbusAddress = 10256; Command_read_regs = Read holding Registers  (0x03); Visibility = No}
    panTimeToOpenCloseValve AT %ID8.2.12.0 [FloatInput]
  Register input module [ID2003] node 13, in %IB8.2.13 out %QB8.2.13 {ModbusAddress = 10258; Command_read_regs = Read holding Registers  (0x03); Visibility = No}
    panMaxTemperature AT %IW8.2.13.0 [WordInput]
  Register input module [ID2003] node 14, in %IB8.2.14 out %QB8.2.14 {ModbusAddress = 10259; Command_read_regs = Read holding Registers  (0x03); Visibility = No}
    panMinTemperature AT %IW8.2.14.0 [WordInput]
  Real input module [ID2007] node 15, in %IB8.2.15 out %QB8.2.15 {ModbusAddress = 10260; Command_read_regs = Read holding Registers  (0x03); Visibility = No}
    panND0502setMaxDosVal AT %ID8.2.15.0 [FloatInput]
  Real input module [ID2007] node 16, in %IB8.2.16 out %QB8.2.16 {ModbusAddress = 10262; Command_read_regs = Read holding Registers  (0x03); Visibility = No}
    panND0502setKoefProp AT %ID8.2.16.0 [FloatInput]
  Real input module [ID2007] node 17, in %IB8.2.17 out %QB8.2.17 {ModbusAddress = 10264; Command_read_regs = Read holding Registers  (0x03); Visibility = No}
    panND0602setMaxDosVal AT %ID8.2.17.0 [FloatInput]
  Real input module [ID2007] node 18, in %IB8.2.18 out %QB8.2.18 {ModbusAddress = 10266; Command_read_regs = Read holding Registers  (0x03); Visibility = No}
    panND0602setKoefProp AT %ID8.2.18.0 [FloatInput]
  Real input module [ID2007] node 19, in %IB8.2.19 out %QB8.2.19 {ModbusAddress = 10268; Command_read_regs = Read holding Registers  (0x03); Visibility = No}
    panND0603setMaxDosVal AT %ID8.2.19.0 [FloatInput]
  Real input module [ID2007] node 20, in %IB8.2.20 out %QB8.2.20 {ModbusAddress = 10270; Command_read_regs = Read holding Registers  (0x03); Visibility = No}
    panND0603setKoefProp AT %ID8.2.20.0 [FloatInput]
  Real input module [ID2007] node 21, in %IB8.2.21 out %QB8.2.21 {ModbusAddress = 10272; Command_read_regs = Read holding Registers  (0x03); Visibility = No}
    panND0703pHsetValue AT %ID8.2.21.0 [FloatInput]
  Real input module [ID2007] node 22, in %IB8.2.22 out %QB8.2.22 {ModbusAddress = 10274; Command_read_regs = Read holding Registers  (0x03); Visibility = No}
    panND0703YoutManual AT %ID8.2.22.0 [FloatInput]
  Real input module [ID2007] node 23, in %IB8.2.23 out %QB8.2.23 {ModbusAddress = 10276; Command_read_regs = Read holding Registers  (0x03); Visibility = No}
    panND0703koeffI AT %ID8.2.23.0 [FloatInput]
  Real input module [ID2007] node 24, in %IB8.2.24 out %QB8.2.24 {ModbusAddress = 10278; Command_read_regs = Read holding Registers  (0x03); Visibility = No}
    panND0703koeffD AT %ID8.2.24.0 [FloatInput]
  Real input module [ID2007] node 25, in %IB8.2.25 out %QB8.2.25 {ModbusAddress = 10280; Command_read_regs = Read holding Registers  (0x03); Visibility = No}
    panND0703koeffP AT %ID8.2.25.0 [FloatInput]
  Real input module [ID2007] node 26, in %IB8.2.26 out %QB8.2.26 {ModbusAddress = 10282; Command_read_regs = Read holding Registers  (0x03); Visibility = No}
    panND0803setMaxDosVal AT %ID8.2.26.0 [FloatInput]
  Real input module [ID2007] node 27, in %IB8.2.27 out %QB8.2.27 {ModbusAddress = 10284; Command_read_regs = Read holding Registers  (0x03); Visibility = No}
    panND0803setKoefProp AT %ID8.2.27.0 [FloatInput]
  Register input module [ID2003] node 28, in %IB8.2.28 out %QB8.2.28 {ModbusAddress = 10286; Command_read_regs = Read holding Registers  (0x03); Visibility = No}
    panND0804doseValue AT %IW8.2.28.0 [WordInput]
  Real input module [ID2007] node 29, in %IB8.2.29 out %QB8.2.29 {ModbusAddress = 10287; Command_read_regs = Read holding Registers  (0x03); Visibility = No}
    panN0105flowSetValue AT %ID8.2.29.0 [FloatInput]
  Real input module [ID2007] node 30, in %IB8.2.30 out %QB8.2.30 {ModbusAddress = 10289; Command_read_regs = Read holding Registers  (0x03); Visibility = No}
    panN0105YoutManual AT %ID8.2.30.0 [FloatInput]
  Real input module [ID2007] node 31, in %IB8.2.31 out %QB8.2.31 {ModbusAddress = 10291; Command_read_regs = Read holding Registers  (0x03); Visibility = No}
    panN0105koeffI AT %ID8.2.31.0 [FloatInput]
  Real input module [ID2007] node 32, in %IB8.2.32 out %QB8.2.32 {ModbusAddress = 10293; Command_read_regs = Read holding Registers  (0x03); Visibility = No}
    panN0105koeffD AT %ID8.2.32.0 [FloatInput]
  Real input module [ID2007] node 33, in %IB8.2.33 out %QB8.2.33 {ModbusAddress = 10295; Command_read_regs = Read holding Registers  (0x03); Visibility = No}
    panN0105koeffP AT %ID8.2.33.0 [FloatInput]
  Real input module [ID2007] node 34, in %IB8.2.34 out %QB8.2.34 {ModbusAddress = 10297; Command_read_regs = Read holding Registers  (0x03); Visibility = No}
    panFQS0301impulsValue AT %ID8.2.34.0 [FloatInput]
  Real input module [ID2007] node 35, in %IB8.2.35 out %QB8.2.35 {ModbusAddress = 10299; Command_read_regs = Read holding Registers  (0x03); Visibility = No}
    panFQS0301correction AT %ID8.2.35.0 [FloatInput]
  Real input module [ID2007] node 36, in %IB8.2.36 out %QB8.2.36 {ModbusAddress = 10301; Command_read_regs = Read holding Registers  (0x03); Visibility = No}
    panFPKtimeToWork AT %ID8.2.36.0 [FloatInput]
  Real input module [ID2007] node 37, in %IB8.2.37 out %QB8.2.37 {ModbusAddress = 10303; Command_read_regs = Read holding Registers  (0x03); Visibility = No}
    panFPKnotStartedTime AT %ID8.2.37.0 [FloatInput]
  Real input module [ID2007] node 38, in %IB8.2.38 out %QB8.2.38 {ModbusAddress = 10305; Command_read_regs = Read holding Registers  (0x03); Visibility = No}
    panFPKmaxPressureValue AT %ID8.2.38.0 [FloatInput]
  Real input module [ID2007] node 39, in %IB8.2.39 out %QB8.2.39 {ModbusAddress = 10307; Command_read_regs = Read holding Registers  (0x03); Visibility = No}
    panFilterValueToRegen AT %ID8.2.39.0 [FloatInput]
ModBus (slave) [MODBUS_ID400] node 9, in %IB9 out %QB9 {SlaveIdentificator = 1; Visibility = No}
  Modbus [MODBUS_ID302] node 0, in %IB9.0 out %QB9.0
    TCP [TCP_ID221] node 0, in %IB9.0.0 out %QB9.0.0 {RemotePort = 502; Visibility = No}
  Float [Float] node 1, in %IB9.1 out %QB9.1
    remFT0101value AT %QD9.1.0 [FloatOutput] Расходомер на входе
  Float [Float] node 2, in %IB9.2 out %QB9.2
    remFQS0301totalAmount AT %QD9.2.0 [FloatOutput] Счетчик очищенных стоков
  Float [Float] node 3, in %IB9.3 out %QB9.3
    remTemperatureValue AT %QD9.3.0 [FloatOutput] Температура в помещении
  8 bits [8Bit] node 4, in %IB9.4 out %QB9.4
    AT %QB9.4.0 [ByteOutput]
  8 bits [8Bit] node 5, in %IB9.5 out %QB9.5
    AT %QB9.5.0 [ByteOutput]
*)

(* POU PLC_PRG, CFC *)
PROGRAM PLC_PRG
VAR

END_VAR
_CFC_ (* Continuous Function Chart, elements in execution order *)
_END_CFC_
END_PROGRAM

(* POU ChoosePumpRegime, CFC *)
FUNCTION_BLOCK ChoosePumpRegime
VAR
	pump1RStrig: RS;		(*Триггер-защелка выбора режима с главным первым насосом.*)
	pump2RStrig: RS;		(*Триггер-защелка выбора режима с главным вторым насосом.*)
	byCounterRStrig: RS;		(*Триггер-защелка выбора режима с запуском по количеству включений.*)
	byWorkTimeRStrig: RS;		(*Триггер-защелка выбора режима с запуском по наработке.*)
	Pump1MainDetector: R_TRIG;		(*Детектор переднего фронта включения режима, когда главный насос - первый.
Для сброса остальных значений.*)
	Pump2MainDetector: R_TRIG;		(*Детектор переднего фронта включения режима, когда главный насос - второй.
Для сброса остальных значений.*)
	ByCounterDetector: R_TRIG;		(*Детектор переднего фронта включения режима по количеству включений.
Для сброса остальных значений.*)
	ByWorkTimeDetector: R_TRIG;		(*Детектор переднего фронта включения режима по наработке.
Для сброса остальных значений.*)
END_VAR
VAR_INPUT
	start: BOOL;		(*Сигнал на включение насоса.
Активируется выход согласно выбранного режима.*)
	pump1Main: BOOL;		(*Режим: первый насос главный, второй - резервный.
Включать импульсом. Включать импульсом.*)
	pump2Main: BOOL;		(*Режим: второй насос главный, первый - резервный.
Включать импульсом. Включать импульсом.*)
	byCounter: BOOL;		(*Режим: запуск по количеству включений.
Включится с меньшим количеством стартов. Включать импульсом.*)
	byWorkTime: BOOL;		(*Режим: запуск по наработке.
Включится насос с меньшей наработкой. Включать импульсом.*)
END_VAR
VAR_OUTPUT
	pump1MainActive: BOOL;		(*Активный режим: первый насос главный.*)
	pump2MainActive: BOOL;		(*Активный режим: второй насос главный.*)
	byCounterActive: BOOL;		(*Активный режим: включение по количеству запусков.*)
	byWorkTimeActive: BOOL;		(*Активный режим: по наработке.*)
	startPump1: BOOL;		(*Запуск первого насоса как главного (основного).*)
	startPump2: BOOL;		(*Запуск второго насоса как главного (основного).*)
	startByCounter: BOOL;		(*Запуск насоса по количеству стартов.
			Запустится с меньшим. Если одинаково, то - первый.*)
	startByWorkTime: BOOL;		(*Запуск по наработке.
			Включится с меньшей. Если одинаково, то - первый.*)
END_VAR
VAR (* helpers for the ST form of the networks *)
	_en62 : BOOL;
	_t62 : BOOL;
	_en72 : BOOL;
	_t72 : BOOL;
	_en78 : BOOL;
	_t78 : BOOL;
	_en84 : BOOL;
	_t84 : BOOL;
END_VAR
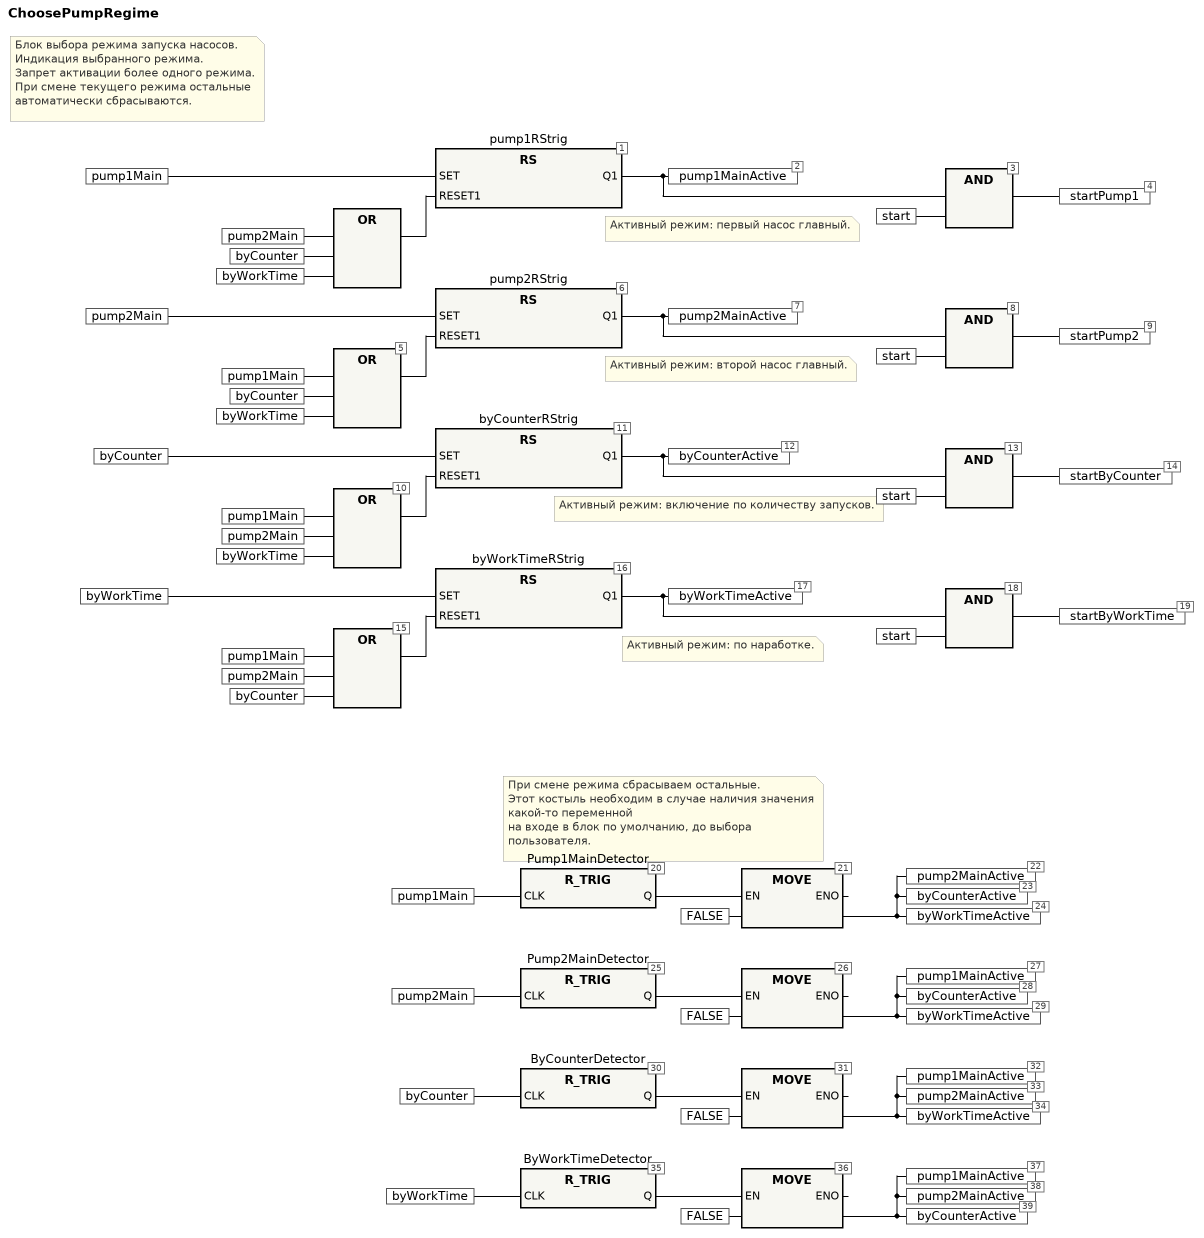
_CFC_ (* Continuous Function Chart, elements in execution order *)
(* При смене режима сбрасываем остальные. / Этот костыль необходим в случае наличия значения какой-то переменной / на входе в блок по умолчанию, до выбора пользователя. *)
(* Активный режим: второй насос главный. *)
(* Активный режим: по наработке. *)
(* Активный режим: включение по количеству запусков. *)
(* Активный режим: первый насос главный. *)
(* Блок выбора режима запуска насосов. / Индикация выбранного режима. / Запрет активации более одного режима. / При смене текущего режима остальные автоматически сбрасываются. *)
#0 OR(pump2Main, byCounter, byWorkTime)
#1 pump1RStrig:RS(SET: pump1Main, RESET1: #0)
#2 pump1MainActive <= #1.Q1
#3 AND(#1.Q1, start)
#4 startPump1 <= #3
#5 OR(pump1Main, byCounter, byWorkTime)
#6 pump2RStrig:RS(SET: pump2Main, RESET1: #5)
#7 pump2MainActive <= #6.Q1
#8 AND(#6.Q1, start)
#9 startPump2 <= #8
#10 OR(pump1Main, pump2Main, byWorkTime)
#11 byCounterRStrig:RS(SET: byCounter, RESET1: #10)
#12 byCounterActive <= #11.Q1
#13 AND(#11.Q1, start)
#14 startByCounter <= #13
#15 OR(pump1Main, pump2Main, byCounter)
#16 byWorkTimeRStrig:RS(SET: byWorkTime, RESET1: #15)
#17 byWorkTimeActive <= #16.Q1
#18 AND(#16.Q1, start)
#19 startByWorkTime <= #18
#20 Pump1MainDetector:R_TRIG(CLK: pump1Main)
#21 MOVE(EN: #20.Q, FALSE)
#22 pump2MainActive <= #21
#23 byCounterActive <= #21
#24 byWorkTimeActive <= #21
#25 Pump2MainDetector:R_TRIG(CLK: pump2Main)
#26 MOVE(EN: #25.Q, FALSE)
#27 pump1MainActive <= #26
#28 byCounterActive <= #26
#29 byWorkTimeActive <= #26
#30 ByCounterDetector:R_TRIG(CLK: byCounter)
#31 MOVE(EN: #30.Q, FALSE)
#32 pump1MainActive <= #31
#33 pump2MainActive <= #31
#34 byWorkTimeActive <= #31
#35 ByWorkTimeDetector:R_TRIG(CLK: byWorkTime)
#36 MOVE(EN: #35.Q, FALSE)
#37 pump1MainActive <= #36
#38 pump2MainActive <= #36
#39 byCounterActive <= #36
_END_CFC_
(* the same logic as Structured Text *)
(* При смене режима сбрасываем остальные. / Этот костыль необходим в случае наличия значения какой-то переменной / на входе в блок по умолчанию, до выбора пользователя. *)
(* Активный режим: второй насос главный. *)
(* Активный режим: по наработке. *)
(* Активный режим: включение по количеству запусков. *)
(* Активный режим: первый насос главный. *)
(* Блок выбора режима запуска насосов. / Индикация выбранного режима. / Запрет активации более одного режима. / При смене текущего режима остальные автоматически сбрасываются. *)
pump1RStrig(SET := pump1Main, RESET1 := pump2Main OR byCounter OR byWorkTime);
pump1MainActive := pump1RStrig.Q1;
startPump1 := pump1RStrig.Q1 AND start;
pump2RStrig(SET := pump2Main, RESET1 := pump1Main OR byCounter OR byWorkTime);
pump2MainActive := pump2RStrig.Q1;
startPump2 := pump2RStrig.Q1 AND start;
byCounterRStrig(SET := byCounter, RESET1 := pump1Main OR pump2Main OR byWorkTime);
byCounterActive := byCounterRStrig.Q1;
startByCounter := byCounterRStrig.Q1 AND start;
byWorkTimeRStrig(SET := byWorkTime, RESET1 := pump1Main OR pump2Main OR byCounter);
byWorkTimeActive := byWorkTimeRStrig.Q1;
startByWorkTime := byWorkTimeRStrig.Q1 AND start;
Pump1MainDetector(CLK := pump1Main);
_en62 := Pump1MainDetector.Q;
IF _en62 THEN _t62 := FALSE; END_IF;
IF _en62 THEN pump2MainActive := _t62; END_IF;
IF _en62 THEN byCounterActive := _t62; END_IF;
IF _en62 THEN byWorkTimeActive := _t62; END_IF;
Pump2MainDetector(CLK := pump2Main);
_en72 := Pump2MainDetector.Q;
IF _en72 THEN _t72 := FALSE; END_IF;
IF _en72 THEN pump1MainActive := _t72; END_IF;
IF _en72 THEN byCounterActive := _t72; END_IF;
IF _en72 THEN byWorkTimeActive := _t72; END_IF;
ByCounterDetector(CLK := byCounter);
_en78 := ByCounterDetector.Q;
IF _en78 THEN _t78 := FALSE; END_IF;
IF _en78 THEN pump1MainActive := _t78; END_IF;
IF _en78 THEN pump2MainActive := _t78; END_IF;
IF _en78 THEN byWorkTimeActive := _t78; END_IF;
ByWorkTimeDetector(CLK := byWorkTime);
_en84 := ByWorkTimeDetector.Q;
IF _en84 THEN _t84 := FALSE; END_IF;
IF _en84 THEN pump1MainActive := _t84; END_IF;
IF _en84 THEN pump2MainActive := _t84; END_IF;
IF _en84 THEN byCounterActive := _t84; END_IF;
END_FUNCTION_BLOCK

(* POU ControlAI, CFC *)
FUNCTION_BLOCK ControlAI
VAR_INPUT
	in: REAL;		(*Входное значение.*)
	minValue: REAL := 0;		(*Минимальное значение на выходе при 4мА на входе.
Если ко входу ничего не подключено, то 0.*)
	maxValue: REAL;		(*Максимальное значение на выходе при 20мА на входе.*)
END_VAR
VAR_OUTPUT
	out: REAL;		(*Выходное отфильтрованное значение.*)
	error: BOOL;		(*Ошибка входа.*)
END_VAR
VAR
	LIN_TRAFO: LIN_TRAFO;		(*Блок масштабирования входной величины.*)
	FilterREAL: FilterREAL;		(*Модуль фильтрации сигнала типа REAL.*)
END_VAR
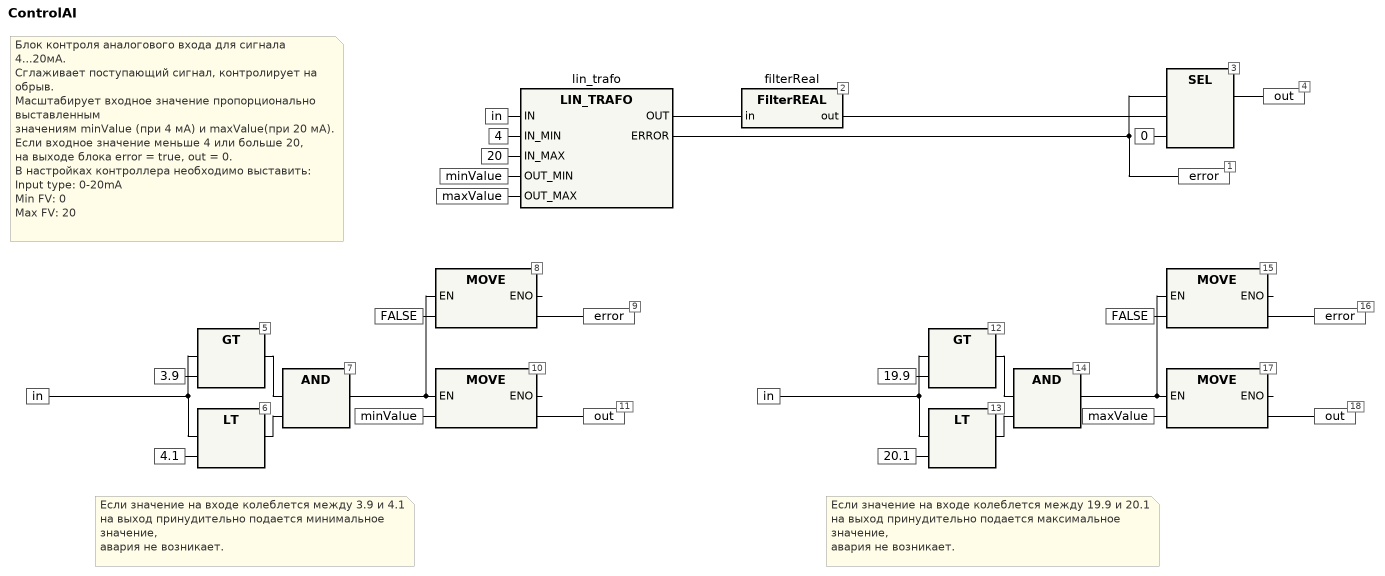
_CFC_ (* Continuous Function Chart, elements in execution order *)
(* Если значение на входе колеблется между 19.9 и 20.1 / на выход принудительно подается максимальное значение, / авария не возникает. *)
(* Если значение на входе колеблется между 3.9 и 4.1 / на выход принудительно подается минимальное значение, / авария не возникает. *)
(* Блок контроля аналогового входа для сигнала 4...20мА. / Сглаживает поступающий сигнал, контролирует на обрыв. / Масштабирует входное значение пропорционально выставленным / значениям minValue (при 4 мА) и maxValue(при 20 мА). / Если входное значение меньше 4 или больше 20, / на выходе блока error = true, out = 0. / В настройках контроллера необходимо выставить: / Input type: 0-20mA / Min FV: 0 / Max FV: 20 *)
#0 lin_trafo:LIN_TRAFO(IN: in, IN_MIN: 4, IN_MAX: 20, OUT_MIN: minValue, OUT_MAX: maxValue)
#1 error <= #0.ERROR
#2 filterReal:FilterREAL(in: #0.OUT)
#3 SEL(#0.ERROR, #2.out, 0)
#4 out <= #3
#5 GT(in, 3.9)
#6 LT(in, 4.1)
#7 AND(#5, #6)
#8 MOVE(EN: #7, FALSE)
#9 error <= #8
#10 MOVE(EN: #7, minValue)
#11 out <= #10
#12 GT(in, 19.9)
#13 LT(in, 20.1)
#14 AND(#12, #13)
#15 MOVE(EN: #14, FALSE)
#16 error <= #15
#17 MOVE(EN: #14, maxValue)
#18 out <= #17
_END_CFC_
END_FUNCTION_BLOCK

(* POU FilterREAL, ST *)
FUNCTION_BLOCK FilterREAL
VAR_INPUT
	in: REAL; (*Входное значение*)
END_VAR
VAR_OUTPUT
	out: REAL; (*Выходное значение*)
END_VAR
VAR
	k: REAL; (*Коэффициент фильтра.Чем меньше тем плавнее, чем больше, тем быстрее работает фильтр.*)
END_VAR
(*Если разница между входом и выходом больше 0,5, то коэффициент большой, фильтр - быстрый, сглаживание - минимально.*)
IF ABS(in - out) > 0.01 THEN
	k := 0.9;
ELSE
	k:=0.0001;
END_IF
out := (in - out) * k + out;
END_FUNCTION_BLOCK

(* POU CounterManager, CFC *)
FUNCTION_BLOCK CounterManager

VAR
	pump1startsCounter: ImpulsCounter;		(*Счетчик количества включений насоса 1.*)
	pump2startsCounter: ImpulsCounter;		(*Счетчик количества включений насоса 2.*)
	counterRtrig: R_TRIG;		(*Детектор переднего фронта сигнала на запуск.*)
	counterFtrig: F_TRIG;		(*Детектор спада сигнала на запуск.*)
	counterRStrigPump1: RS;		(*RSтриггер сигнала на запуск насоса 1.*)
	counterRStrigPump2: RS;		(*RSтриггер сигнала на запуск насоса 2.*)
END_VAR
VAR_INPUT
	counterStart: BOOL;		(*Сигнал на запуск насоса с наименьшей наработкой.*)
	pump1ON: BOOL;		(*Сигнал подтверждение о запуске насоса 1.*)
	pump2ON: BOOL;		(*Сигнал подтверждение о запуске насоса 2.*)
	Pump1ResetCounter: BOOL;		(*Сброс счетчика включений насоса 1.*)
	Pump2ResetCounter: BOOL;		(*Сброс счетчика включений насоса 2.*)
END_VAR
VAR_OUTPUT
	counterPump1ON: BOOL;		(*Сигнал на запуск насоса 1.*)
	counterPump2ON: BOOL;		(*Сигнал на запуск насоса 2.*)
	counterPump1: DWORD;		(*Количество включений насоса 1.*)
	counterPump2: DWORD;		(*Количество включений насоса 2.*)
END_VAR
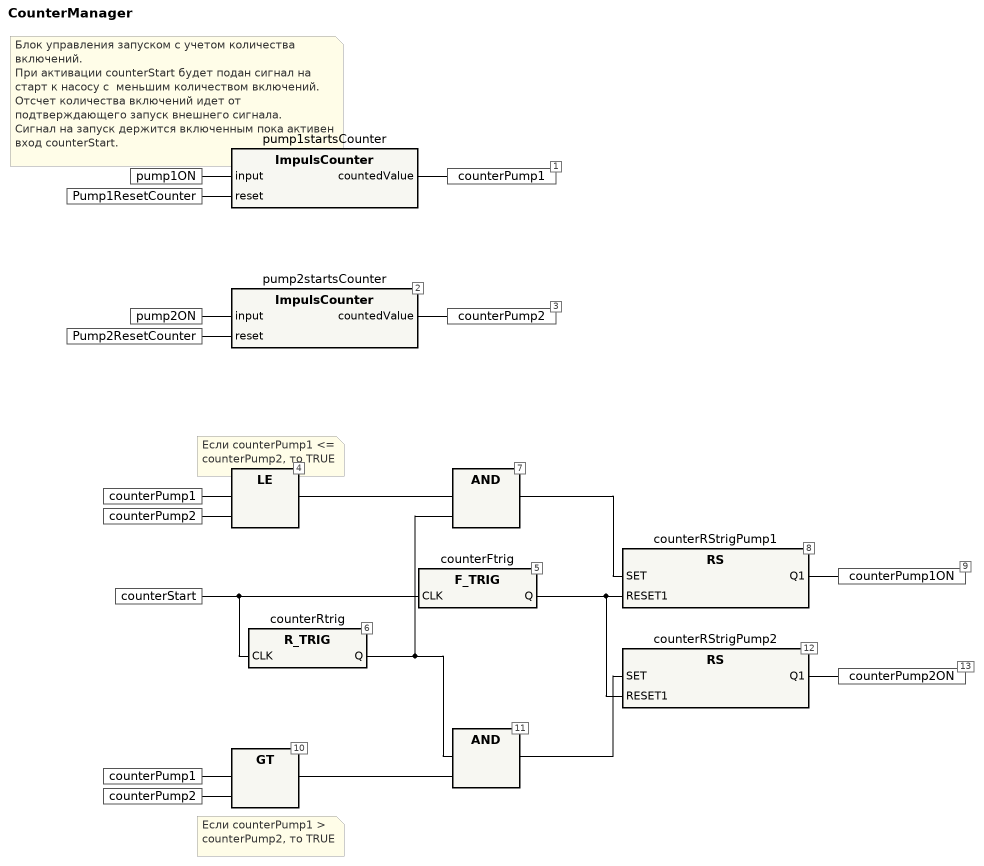
_CFC_ (* Continuous Function Chart, elements in execution order *)
(* Блок управления запуском с учетом количества включений. / При активации counterStart будет подан сигнал на старт к насосу с  меньшим количеством включений. / Отсчет количества включений идет от подтверждающего запуск внешнего сигнала. / Сигнал на запуск держится включенным пока активен вход counterStart. *)
(* Если counterPump1 <= / counterPump2, то TRUE *)
(* Если counterPump1 > / counterPump2, то TRUE *)
#0 pump1startsCounter:ImpulsCounter(input: pump1ON, reset: Pump1ResetCounter)
#1 counterPump1 <= #0.countedValue
#2 pump2startsCounter:ImpulsCounter(input: pump2ON, reset: Pump2ResetCounter)
#3 counterPump2 <= #2.countedValue
#4 LE(counterPump1, counterPump2)
#5 counterFtrig:F_TRIG(CLK: counterStart)
#6 counterRtrig:R_TRIG(CLK: counterStart)
#7 AND(#4, #6.Q)
#8 counterRStrigPump1:RS(SET: #7, RESET1: #5.Q)
#9 counterPump1ON <= #8.Q1
#10 GT(counterPump1, counterPump2)
#11 AND(#6.Q, #10)
#12 counterRStrigPump2:RS(SET: #11, RESET1: #5.Q)
#13 counterPump2ON <= #12.Q1
_END_CFC_
END_FUNCTION_BLOCK

(* POU ImpulsCounter, CFC *)
FUNCTION_BLOCK ImpulsCounter
VAR
	ImpulsDetector: R_TRIG;		(*Триггер переднего фронта входящего импульса.*)
END_VAR
VAR_INPUT
	input: BOOL;		(*Вход для импульсов, которые надо сосчитать.*)
	reset: BOOL;		(*Сброс счетчика.*)
END_VAR
VAR_OUTPUT
	countedValue: DWORD;		(*Суммарное количество импульсов.*)
END_VAR
VAR (* helpers for the ST form of the networks *)
	_t8 : DWORD;
END_VAR
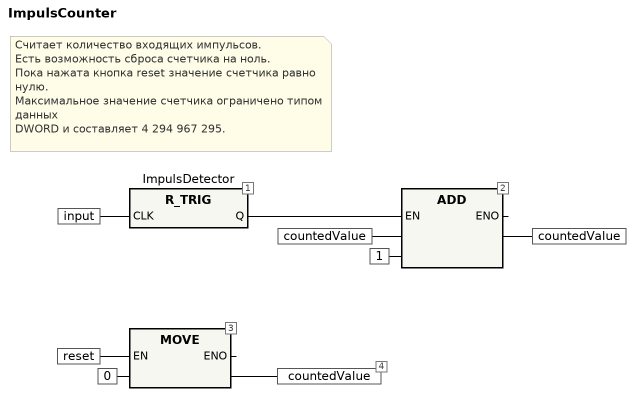
_CFC_ (* Continuous Function Chart, elements in execution order *)
(* Считает количество входящих импульсов. / Есть возможность сброса счетчика на ноль. / Пока нажата кнопка reset значение счетчика равно нулю. / Максимальное значение счетчика ограничено типом данных / DWORD и составляет 4 294 967 295. *)
#0 countedValue <= #2
#1 ImpulsDetector:R_TRIG(CLK: input)
#2 ADD(EN: #1.Q, countedValue, 1)
#3 MOVE(EN: reset, 0)
#4 countedValue <= #3
_END_CFC_
(* the same logic as Structured Text *)
(* Считает количество входящих импульсов. / Есть возможность сброса счетчика на ноль. / Пока нажата кнопка reset значение счетчика равно нулю. / Максимальное значение счетчика ограничено типом данных / DWORD и составляет 4 294 967 295. *)
countedValue := _t8;
ImpulsDetector(CLK := input);
IF ImpulsDetector.Q THEN _t8 := countedValue + 1; END_IF;
IF reset THEN countedValue := 0; END_IF;
END_FUNCTION_BLOCK

(* POU DosingPumpProportional, CFC *)
FUNCTION_BLOCK DosingPumpProportional
VAR_INPUT
	flowValue: REAL;		(*текущее значение мгновенного расхода, кубометров в час.*)
	setMinPumpDosingValue: REAL := 0;		(*задание минимальной производительности доз.насоса.
По умолчанию, если ничего не подключено ко входу, равно нулю.*)
	setMaxPumpDosingValue: REAL;		(*задание максимальной производительности доз.насоса, в мл/мин*)
	minOutputValue: REAL := 4;		(*минимальное значение выходного сигнала.
По умолчанию, если ничего не подключено ко входу, равно 4.*)
	maxOutputValue: REAL := 20;		(*Максимально значение выходного сигнала.
По умолчанию, если ничего не подключено ко входу, равно 20.*)
	setKoeffProportionality: REAL;		(*Задание мл на кубометр (коэф.пропорциональности между расходом и дозированием)*)
	minFlowToStart: REAL := 10;		(*Минимальное значение расхода для подачи сигнала на начало дозирования.
По умолчанию, если ничего не подключено ко входу, равно 10 кубометров в час.*)
END_VAR
VAR_OUTPUT
	outputValue: REAL;		(*Выходной сигнал на дозирующий насос.*)
	dosingError: BOOL;		(*Ошибка производительности дозирования (неверно заданы значения производительности насоса, производительность доз.насоса не соответствует расходу.*)
	startDosingPump: BOOL;		(*Сигнал на запуск дозирующего насоса.*)
END_VAR
VAR
	linearTransformator: LIN_TRAFO;		(*получает на вход значение из указанного диапазона, ставит на выходе пропорциональное значение из другого диапазона.*)
END_VAR
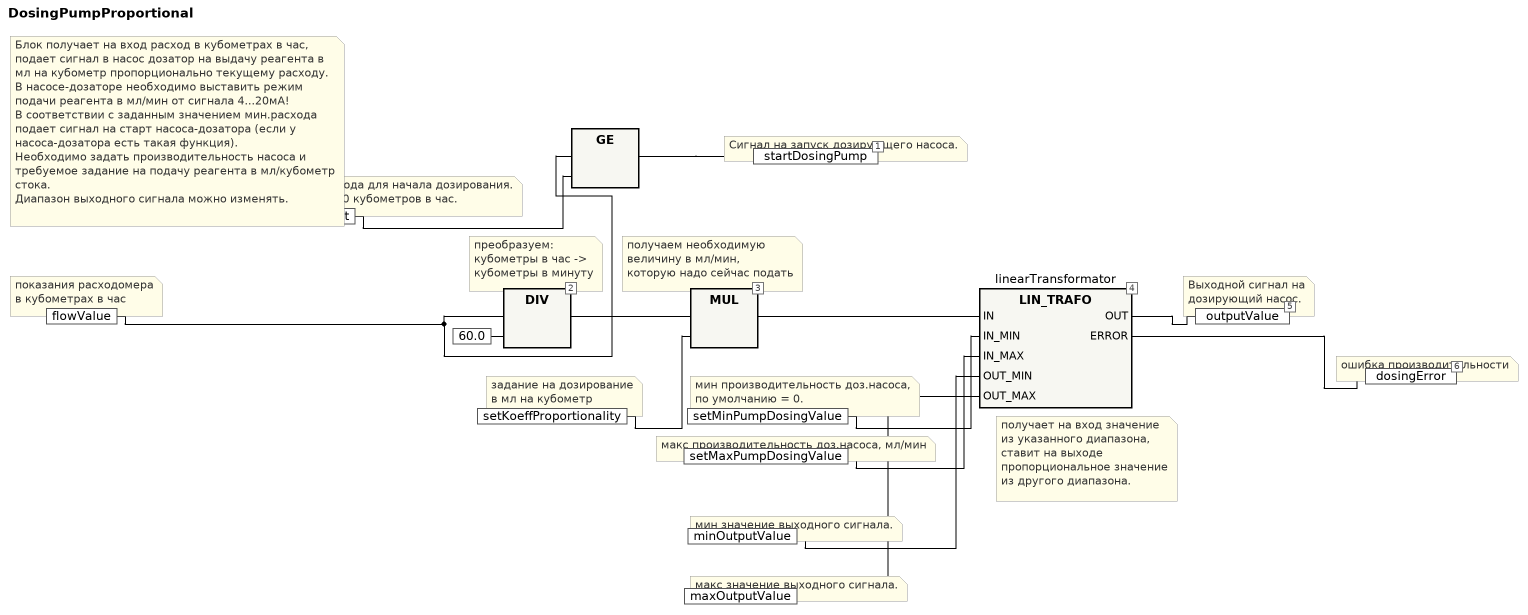
_CFC_ (* Continuous Function Chart, elements in execution order *)
(* Сигнал на запуск дозирующего насоса. *)
(* min значение расхода для начала дозирования. / По умолчанию = 10 кубометров в час. *)
(* макс производительность доз.насоса, мл/мин *)
(* мин производительность доз.насоса, / по умолчанию = 0. *)
(* получаем необходимую / величину в мл/мин, / которую надо сейчас подать *)
(* задание на дозирование / в мл на кубометр *)
(* показания расходомера / в кубометрах в час *)
(* преобразуем: / кубометры в час -> / кубометры в минуту *)
(* мин значение выходного сигнала. *)
(* макс значение выходного сигнала. *)
(* Выходной сигнал на / дозирующий насос. *)
(* ошибка производительности *)
(* получает на вход значение / из указанного диапазона, / ставит на выходе / пропорциональное значение / из другого диапазона. *)
(* Блок получает на вход расход в кубометрах в час, подает сигнал в насос дозатор на выдачу реагента в мл на кубометр пропорционально текущему расходу. / В насосе-дозаторе необходимо выставить режим подачи реагента в мл/мин от сигнала 4...20мА! / В соответствии с заданным значением мин.расхода подает сигнал на старт насоса-дозатора (если у насоса-дозатора есть такая функция). / Необходимо задать производительность насоса и требуемое задание на подачу реагента в мл/кубометр стока. / Диапазон выходного сигнала можно изменять. *)
#0 GE(flowValue, minFlowToStart)
#1 startDosingPump <= #0
#2 DIV(flowValue, 60.0)
#3 MUL(#2, setKoeffProportionality)
#4 linearTransformator:LIN_TRAFO(IN: #3, IN_MIN: setMinPumpDosingValue, IN_MAX: setMaxPumpDosingValue, OUT_MIN: minOutputValue, OUT_MAX: maxOutputValue)
#5 outputValue <= #4.OUT
#6 dosingError <= #4.ERROR
_END_CFC_
(* the same logic as Structured Text *)
(* Сигнал на запуск дозирующего насоса. *)
(* min значение расхода для начала дозирования. / По умолчанию = 10 кубометров в час. *)
(* макс производительность доз.насоса, мл/мин *)
(* мин производительность доз.насоса, / по умолчанию = 0. *)
(* получаем необходимую / величину в мл/мин, / которую надо сейчас подать *)
(* задание на дозирование / в мл на кубометр *)
(* показания расходомера / в кубометрах в час *)
(* преобразуем: / кубометры в час -> / кубометры в минуту *)
(* мин значение выходного сигнала. *)
(* макс значение выходного сигнала. *)
(* Выходной сигнал на / дозирующий насос. *)
(* ошибка производительности *)
(* получает на вход значение / из указанного диапазона, / ставит на выходе / пропорциональное значение / из другого диапазона. *)
(* Блок получает на вход расход в кубометрах в час, подает сигнал в насос дозатор на выдачу реагента в мл на кубометр пропорционально текущему расходу. / В насосе-дозаторе необходимо выставить режим подачи реагента в мл/мин от сигнала 4...20мА! / В соответствии с заданным значением мин.расхода подает сигнал на старт насоса-дозатора (если у насоса-дозатора есть такая функция). / Необходимо задать производительность насоса и требуемое задание на подачу реагента в мл/кубометр стока. / Диапазон выходного сигнала можно изменять. *)
startDosingPump := flowValue >= minFlowToStart;
linearTransformator(IN := (flowValue / 60.0) * setKoeffProportionality, IN_MIN := setMinPumpDosingValue, IN_MAX := setMaxPumpDosingValue, OUT_MIN := minOutputValue, OUT_MAX := maxOutputValue);
outputValue := linearTransformator.OUT;
dosingError := linearTransformator.ERROR;
END_FUNCTION_BLOCK

(* POU FlowVolume, CFC *)
FUNCTION_BLOCK FlowVolume
VAR_INPUT
	flowValue: REAL;		(*Вход от расходомера, мгновенный расход в кубометрах в час.*)
	setVolume: REAL;		(*Контрольный объем. Сравнивается с накопленным по показаниям расходомера,
Если превышает, счетчик сбрасывается, на выход out подается импульс.
Если на входе ноль, то условие не работает, блок просто считает сумму стоков.*)
	reset: BOOL;		(*Ручной сброс счетчика.*)
END_VAR
VAR_OUTPUT
	totalAmount: REAL;		(*Сумма накопленных стоков.*)
	out: BOOL;		(*Импульс - сигнал что сумма стоков равна или больше
заданному в setVolume значению.*)
END_VAR
VAR
	pulsPerSec: PulsePerSec;		(*Генератор импульс в секунду.*)
END_VAR
VAR (* helpers for the ST form of the networks *)
	_t22 : BOOL;
END_VAR
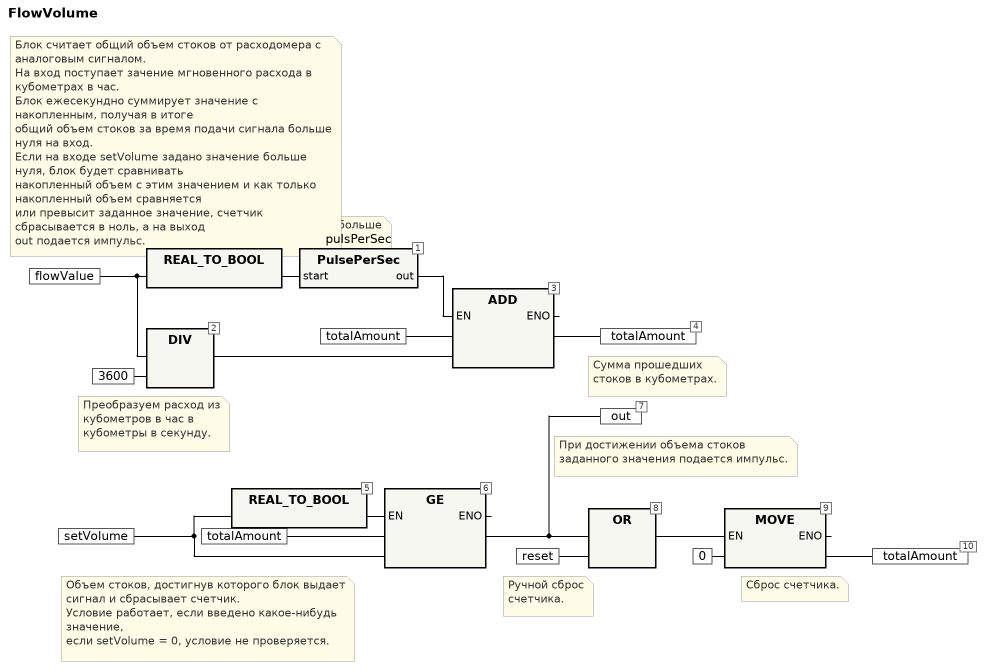
_CFC_ (* Continuous Function Chart, elements in execution order *)
(* Ручной сброс / счетчика. *)
(* При достижении объема стоков / заданного значения подается импульс. *)
(* Сумма прошедших / стоков в кубометрах. *)
(* Объем стоков, достигнув которого блок выдает / сигнал и сбрасывает счетчик. / Условие работает, если введено какое-нибудь значение, / если setVolume = 0, условие не проверяется. *)
(* Преобразуем расход из / кубометров в час в / кубометры в секунду. *)
(* Начинаем считать стоки при наличии расхода больше нуля. *)
(* Сброс счетчика. *)
(* Блок считает общий объем стоков от расходомера с аналоговым сигналом. / На вход поступает зачение мгновенного расхода в кубометрах в час. / Блок ежесекундно суммирует значение с накопленным, получая в итоге / общий объем стоков за время подачи сигнала больше нуля на вход. / Если на входе setVolume задано значение больше нуля, блок будет сравнивать / накопленный объем с этим значением и как только накопленный объем сравняется / или превысит заданное значение, счетчик сбрасывается в ноль, а на выход / out подается импульс. *)
#0 REAL_TO_BOOL(flowValue)
#1 pulsPerSec:PulsePerSec(start: #0)
#2 DIV(flowValue, 3600)
#3 ADD(EN: #1.out, totalAmount, #2)
#4 totalAmount <= #3
#5 REAL_TO_BOOL(setVolume)
#6 GE(EN: #5, totalAmount, setVolume)
#7 out <= #6
#8 OR(#6, reset)
#9 MOVE(EN: #8, 0)
#10 totalAmount <= #9
_END_CFC_
(* the same logic as Structured Text *)
(* Ручной сброс / счетчика. *)
(* При достижении объема стоков / заданного значения подается импульс. *)
(* Сумма прошедших / стоков в кубометрах. *)
(* Объем стоков, достигнув которого блок выдает / сигнал и сбрасывает счетчик. / Условие работает, если введено какое-нибудь значение, / если setVolume = 0, условие не проверяется. *)
(* Преобразуем расход из / кубометров в час в / кубометры в секунду. *)
(* Начинаем считать стоки при наличии расхода больше нуля. *)
(* Сброс счетчика. *)
(* Блок считает общий объем стоков от расходомера с аналоговым сигналом. / На вход поступает зачение мгновенного расхода в кубометрах в час. / Блок ежесекундно суммирует значение с накопленным, получая в итоге / общий объем стоков за время подачи сигнала больше нуля на вход. / Если на входе setVolume задано значение больше нуля, блок будет сравнивать / накопленный объем с этим значением и как только накопленный объем сравняется / или превысит заданное значение, счетчик сбрасывается в ноль, а на выход / out подается импульс. *)
pulsPerSec(start := REAL_TO_BOOL(flowValue));
IF pulsPerSec.out THEN totalAmount := totalAmount + (flowValue / 3600); END_IF;
IF REAL_TO_BOOL(setVolume) THEN _t22 := totalAmount >= setVolume; END_IF;
out := _t22;
IF _t22 OR reset THEN totalAmount := 0; END_IF;
END_FUNCTION_BLOCK

(* POU PulsePerSec, CFC *)
FUNCTION_BLOCK PulsePerSec
VAR_INPUT
	start: BOOL;		(*Включает генератор импульсов.*)
END_VAR
VAR_OUTPUT
	out: BOOL;		(*Выход генератора импульсов. Начинает с FALSE.
			Каждую секунду выдает BOOL: TRUE.*)
END_VAR
VAR
	pulserRtrig: R_TRIG;		(*Детектор переднего фронта подачи импульсов.*)
	pulserRTC: RTC;		(*Таймер реального времени.*)
END_VAR
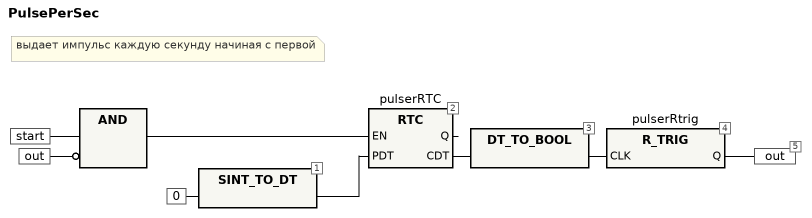
_CFC_ (* Continuous Function Chart, elements in execution order *)
(* выдает импульс каждую секунду начиная с первой *)
#0 AND(start, NOT out)
#1 SINT_TO_DT(0)
#2 pulserRTC:RTC(EN: #0, PDT: #1)
#3 DT_TO_BOOL(#2.CDT)
#4 pulserRtrig:R_TRIG(CLK: #3)
#5 out <= #4.Q
_END_CFC_
(* the same logic as Structured Text *)
(* выдает импульс каждую секунду начиная с первой *)
pulserRTC(EN := start AND NOT out, PDT := SINT_TO_DT(0));
pulserRtrig(CLK := DT_TO_BOOL(pulserRTC.CDT));
out := pulserRtrig.Q;
END_FUNCTION_BLOCK

(* POU IfBOOL, ST *)
FUNCTION_BLOCK IfBOOL
VAR_INPUT
	key: BOOL; (*Ключ. Если TRUE, то сигнал на входе будет передан на выход keyTRUE, иначе на keyFALSE.*)
	input: BOOL; (*Вход*)
END_VAR
VAR_OUTPUT
	keyFALSE: BOOL; (*Выход  получит значение от входа, если key = FALSE.*)
	keyTRUE: BOOL; (*Выход  получит значение от входа, если key = TRUE.*)
END_VAR
VAR
END_VAR
IF key = TRUE THEN
	keyTRUE := input;
	keyFALSE := FALSE;
ELSE keyTRUE := FALSE;
		keyFALSE := input;
END_IF
END_FUNCTION_BLOCK

(* POU ImpulsFlowCounter, CFC *)
FUNCTION_BLOCK ImpulsFlowCounter
VAR_INPUT
	impulsInput: BOOL;		(*Входящие импульсы от расходомера.
Каждый импульс будет прибавлять в итоговую сумму величину веса импульса.*)
	impulsValue: REAL;		(*Вес импульса расходомера.*)
	resetCounter: BOOL;		(*Сброс счетчика.*)
	correctionValue: REAL;		(*Число, которое будет прибавлено или вычтено из накопленной суммы.*)
	addCorrection: BOOL;		(*Прибавить коррекцию к накопленной сумме.*)
	deleteCorrection: BOOL;		(*Вычесть коррекцию из накопленной суммы.
Если получится отрицательное число, сумма скинется в ноль.*)
END_VAR
VAR_OUTPUT
	totalAmountREAL: REAL;		(*Накопленная сумма в десятичном виде.
От 10 млн может выводиться в экспоненциальной форме.*)
	totalAmountDWORD: DWORD;		(*Накопленная сумма в целочисленном виде.
Округление десятичных по правилам арифметики.*)
END_VAR
VAR
	inputImpulsRtrig: R_TRIG;		(*Детектор переднего фронта входящих импульсов.*)
	resetRtrig: R_TRIG;		(*Детектор переднего фронта сигнала на сброс счетчика.*)
	addCorrRtrig: R_TRIG;		(*Детектор переднего фронта сигнала на прибавление коррекции.*)
	deleteCorrRtrig: R_TRIG;		(*Детектор переднего фронта сигнала на вычитание коррекции.*)
END_VAR
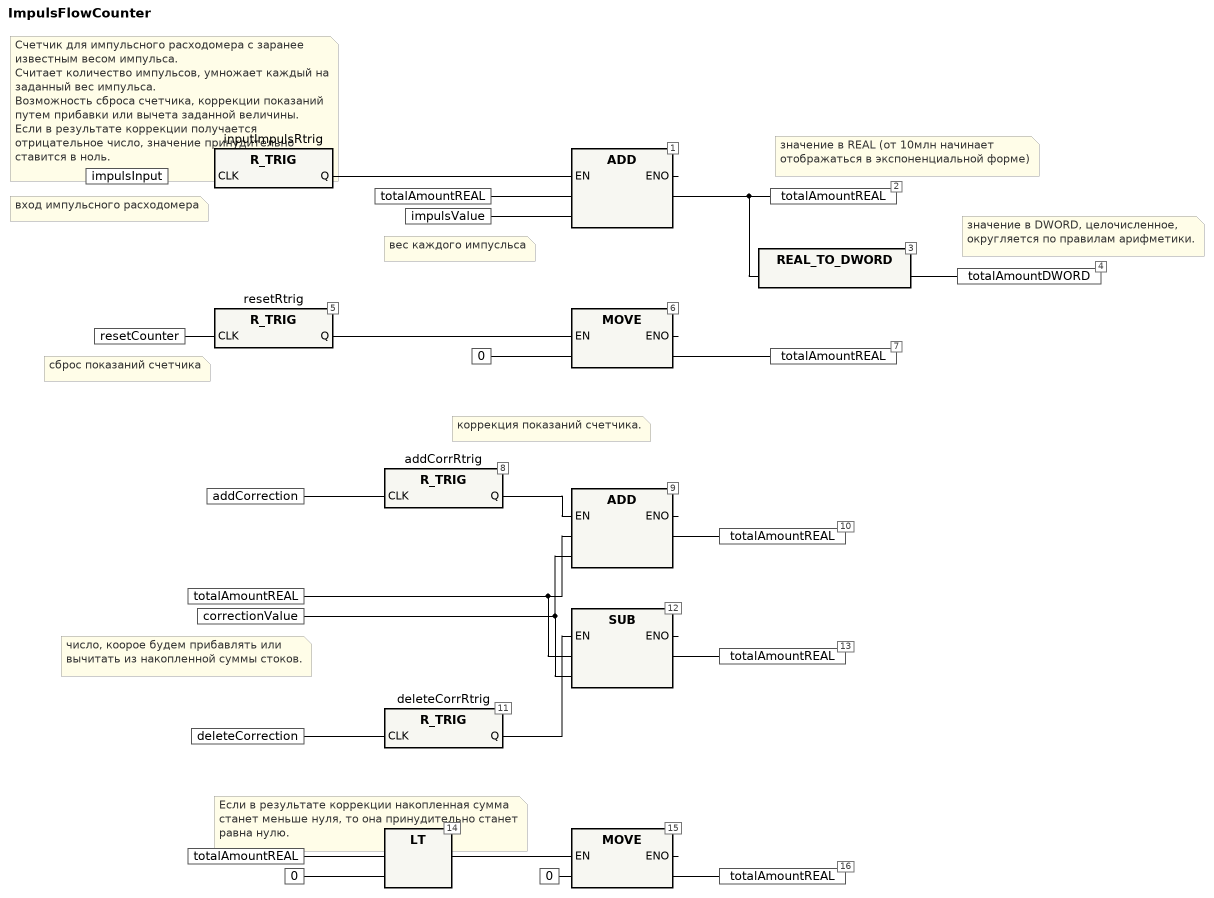
_CFC_ (* Continuous Function Chart, elements in execution order *)
(* вход импульсного расходомера *)
(* сброс показаний счетчика *)
(* значение в REAL (от 10млн начинает / отображаться в экспоненциальной форме) *)
(* значение в DWORD, целочисленное, / округляется по правилам арифметики. *)
(* Если в результате коррекции накопленная сумма станет меньше нуля, то она принудительно станет равна нулю. *)
(* коррекция показаний счетчика. *)
(* число, коорое будем прибавлять или / вычитать из накопленной суммы стоков. *)
(* вес каждого импусльса *)
(* Счетчик для импульсного расходомера с заранее известным весом импульса. / Считает количество импульсов, умножает каждый на заданный вес импульса. / Возможность сброса счетчика, коррекции показаний путем прибавки или вычета заданной величины. / Если в результате коррекции получается отрицательное число, значение принудительно ставится в ноль. *)
#0 inputImpulsRtrig:R_TRIG(CLK: impulsInput)
#1 ADD(EN: #0.Q, totalAmountREAL, impulsValue)
#2 totalAmountREAL <= #1
#3 REAL_TO_DWORD(#1)
#4 totalAmountDWORD <= #3
#5 resetRtrig:R_TRIG(CLK: resetCounter)
#6 MOVE(EN: #5.Q, 0)
#7 totalAmountREAL <= #6
#8 addCorrRtrig:R_TRIG(CLK: addCorrection)
#9 ADD(EN: #8.Q, totalAmountREAL, correctionValue)
#10 totalAmountREAL <= #9
#11 deleteCorrRtrig:R_TRIG(CLK: deleteCorrection)
#12 SUB(EN: #11.Q, totalAmountREAL, correctionValue)
#13 totalAmountREAL <= #12
#14 LT(totalAmountREAL, 0)
#15 MOVE(EN: #14, 0)
#16 totalAmountREAL <= #15
_END_CFC_
END_FUNCTION_BLOCK

(* POU QueueManager, CFC *)
FUNCTION_BLOCK QueueManager
VAR_INPUT
	input: BOOL;		(*Вход сигнала на регенерацию.*)
	testValves: BOOL;		(*Тест заслонок. Имитирует подачу сигнала на регенерацию.*)
	filterAlarm: BOOL;		(*Сигнал авария от управляющего клапана.*)
	regenFilterStatus: BOOL;		(*Сигнал от управляющего клапана о текущем режиме.*)
	alarmReset: BOOL;		(*Сброс аварий.*)
	startNextLoop: BOOL;		(*Запуск нового цикла регенерации. Все сигналы о том, что фильтры
отрегенерированы сбрасываются.*)
	filterValveOpened: BOOL;		(*Заслонка фильтрации открыта.*)
	filterValveClosed: BOOL;		(*Заслонка фильтрации закрыта.*)
	regenValveOpened: BOOL;		(*Заслонка регенерации открыта.*)
	regenValveClosed: BOOL;		(*Заслонка регенерации закрыта.*)
	timeToOpenClose: WORD;		(*Время на открытие/закрытие заслонки в секундах.*)
END_VAR
VAR_OUTPUT
	output: BOOL;		(*Выход для связи с остальными блоками управления очередью
на промывку. В последнем не подключается.*)
	filterValveToOpen: BOOL;		(*Открыть заслонку фильтрации.*)
	filterValveToClose: BOOL;		(*Закрыть заслонку фильтрации.*)
	errorToOpenFilterValve: BOOL;		(*Заслонка фильтрации не открылась за заданное время.*)
	errorToCloseFilterValve: BOOL;		(*Заслонка фильтрации не закрылась за заданное время.*)
	regenValveToOpen: BOOL;		(*Открыть заслонку регенерации.*)
	regenValveToClose: BOOL;		(*Закрыть заслонку регенерации.*)
	errorToOpenRegenValve: BOOL;		(*Заслонка регенерации не открылась за заданное время.*)
	errorToCloseRegenValve: BOOL;		(*Заслонка регенерации не закрылась за заданное время.*)
	regenerated: BOOL;		(*Фильтр прошел регенерацию.*)
	failToRegen: BOOL;		(*Попытка регенерации не удалась.*)
	loopFinished: BOOL;		(*Вход последнего блока подключить во входы startNextLoop во всех блоках,
включая самого себя. В остальных блоках выход не задействовать.*)
	startRegen: BOOL; (*Команда на промывку фильтра*)
END_VAR
VAR
	valveAlarm: BOOL;		(*Общий сигнал авария от обеих заслонок.*)
	QueueModule: QueueModule;		(*Модуль управления очередью на регенерацию.*)
	filterValve: SimpleValve;		(*Блок управления заслонкой фильтрации.*)
	regenrValve: SimpleValve;		(*Блок управления заслонкой регенерации.*)
END_VAR
VAR (* helpers for the ST form of the networks *)
	_t21 : BOOL;
END_VAR
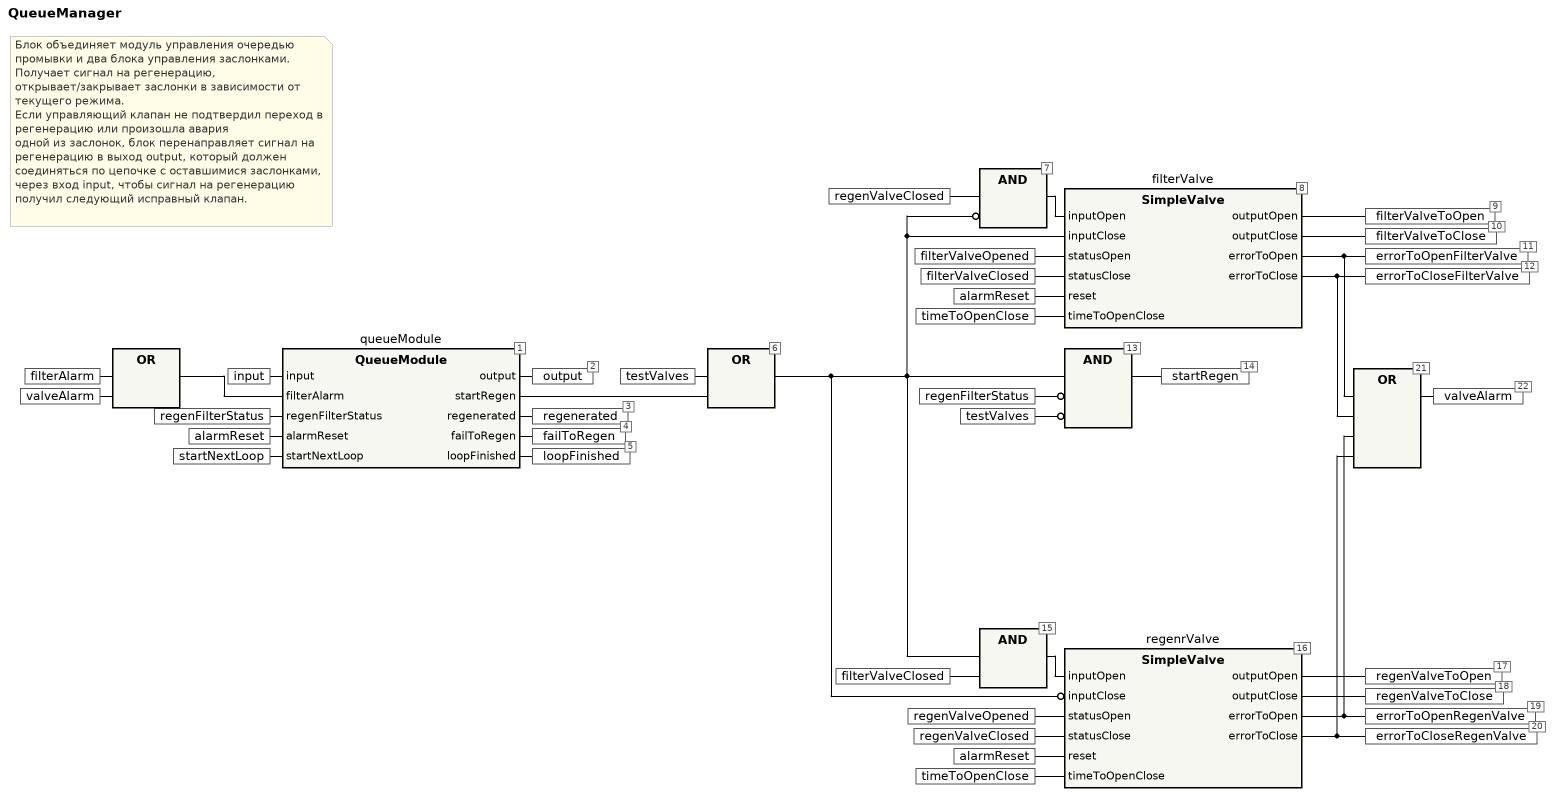
_CFC_ (* Continuous Function Chart, elements in execution order *)
(* Блок объединяет модуль управления очередью промывки и два блока управления заслонками. / Получает сигнал на регенерацию, открывает/закрывает заслонки в зависимости от текущего режима. / Если управляющий клапан не подтвердил переход в регенерацию или произошла авария / одной из заслонок, блок перенаправляет сигнал на регенерацию в выход output, который должен / соединяться по цепочке с оставшимися заслонками, через вход input, чтобы сигнал на регенерацию / получил следующий исправный клапан. *)
#0 OR(filterAlarm, valveAlarm)
#1 queueModule:QueueModule(input: input, filterAlarm: #0, regenFilterStatus: regenFilterStatus, alarmReset: alarmReset, startNextLoop: startNextLoop)
#2 output <= #1.output
#3 regenerated <= #1.regenerated
#4 failToRegen <= #1.failToRegen
#5 loopFinished <= #1.loopFinished
#6 OR(testValves, #1.startRegen)
#7 AND(regenValveClosed, NOT #6)
#8 filterValve:SimpleValve(inputOpen: #7, inputClose: #6, statusOpen: filterValveOpened, statusClose: filterValveClosed, reset: alarmReset, timeToOpenClose: timeToOpenClose)
#9 filterValveToOpen <= #8.outputOpen
#10 filterValveToClose <= #8.outputClose
#11 errorToOpenFilterValve <= #8.errorToOpen
#12 errorToCloseFilterValve <= #8.errorToClose
#13 AND(#6, NOT regenFilterStatus, NOT testValves)
#14 startRegen <= #13
#15 AND(#6, filterValveClosed)
#16 regenrValve:SimpleValve(inputOpen: #15, inputClose: NOT #6, statusOpen: regenValveOpened, statusClose: regenValveClosed, reset: alarmReset, timeToOpenClose: timeToOpenClose)
#17 regenValveToOpen <= #16.outputOpen
#18 regenValveToClose <= #16.outputClose
#19 errorToOpenRegenValve <= #16.errorToOpen
#20 errorToCloseRegenValve <= #16.errorToClose
#21 OR(#8.errorToOpen, #8.errorToClose, #16.errorToOpen, #16.errorToClose)
#22 valveAlarm <= #21
_END_CFC_
(* the same logic as Structured Text *)
(* Блок объединяет модуль управления очередью промывки и два блока управления заслонками. / Получает сигнал на регенерацию, открывает/закрывает заслонки в зависимости от текущего режима. / Если управляющий клапан не подтвердил переход в регенерацию или произошла авария / одной из заслонок, блок перенаправляет сигнал на регенерацию в выход output, который должен / соединяться по цепочке с оставшимися заслонками, через вход input, чтобы сигнал на регенерацию / получил следующий исправный клапан. *)
queueModule(input := input, filterAlarm := filterAlarm OR valveAlarm, regenFilterStatus := regenFilterStatus, alarmReset := alarmReset, startNextLoop := startNextLoop);
output := queueModule.output;
regenerated := queueModule.regenerated;
failToRegen := queueModule.failToRegen;
loopFinished := queueModule.loopFinished;
_t21 := testValves OR queueModule.startRegen;
filterValve(inputOpen := regenValveClosed AND NOT _t21, inputClose := _t21, statusOpen := filterValveOpened, statusClose := filterValveClosed, reset := alarmReset, timeToOpenClose := timeToOpenClose);
filterValveToOpen := filterValve.outputOpen;
filterValveToClose := filterValve.outputClose;
errorToOpenFilterValve := filterValve.errorToOpen;
errorToCloseFilterValve := filterValve.errorToClose;
startRegen := _t21 AND NOT regenFilterStatus AND NOT testValves;
regenrValve(inputOpen := _t21 AND filterValveClosed, inputClose := NOT _t21, statusOpen := regenValveOpened, statusClose := regenValveClosed, reset := alarmReset, timeToOpenClose := timeToOpenClose);
regenValveToOpen := regenrValve.outputOpen;
regenValveToClose := regenrValve.outputClose;
errorToOpenRegenValve := regenrValve.errorToOpen;
errorToCloseRegenValve := regenrValve.errorToClose;
valveAlarm := filterValve.errorToOpen OR filterValve.errorToClose OR regenrValve.errorToOpen OR regenrValve.errorToClose;
END_FUNCTION_BLOCK

(* POU QueueModule, CFC *)
FUNCTION_BLOCK QueueModule
VAR_INPUT
	input: BOOL;		(*Вход на старт регенерации.*)
	filterAlarm: BOOL;		(*Вход аварии от управляющего клапана фильтра.*)
	regenFilterStatus: BOOL;		(*Вход для сигнала подтверждения начала регенерации
от фильтра.*)
	alarmReset: BOOL;		(*Сброс статуса о неудачной попытке регенерации.*)
	startNextLoop: BOOL;		(*Запустить новый цикл, сбрасываются все статусы промытости
фильтров, начало снова от первого фильтра.*)
END_VAR
VAR_OUTPUT
	output: BOOL;		(*Выход, передающий сигнал от счетчика о начале регенерации,
на следующий фильтр. Соединять с input следующего блока, если он есть.*)
	startRegen: BOOL;		(*Выход на старт регенерации, подаваемый на фильтр.*)
	regenerated: BOOL;		(*TRUE, если этот фильтр уже промыт.*)
	failToRegen: BOOL;		(*Не удалось запустить регенерацию.
Не пришло подтверждение от фильтра более 5 сек после старта.*)
	loopFinished: BOOL;		(*Импульсный сигнал, возникающий при отключени сигнала подтверждения
статуса промывки от фильтра (фильтр вернулся в режим фильтрации) или при неудачной попытке регенерации. 
Использовать в последнем блоке для старта нового цикла во всех блоках.*)
END_VAR
VAR
	regStatusDelay: TON;		(*Таймер задержки ожидания подтверждения от фильтра
о начале регенерации.*)
	regStartRS: RS;		(*Триггер старта регенерации.*)
	failureRS: RS;		(*Триггер неудачного пуска регенерации.*)
	successRS: RS;		(*Триггер удачной регенерации.*)
	regenFilterOFF: F_TRIG;		(*Триггер контроля отключения сигнала от фильтра, что он закончил
режим промывки для возврата задвижек обратно в режим фильтрации.*)
	failureRtrig: R_TRIG;		(*детектор переднего фронта сигнала о неудачной попытке регенерации.*)
END_VAR
VAR (* helpers for the ST form of the networks *)
	_t45 : BOOL;
	_t78 : BOOL;
END_VAR
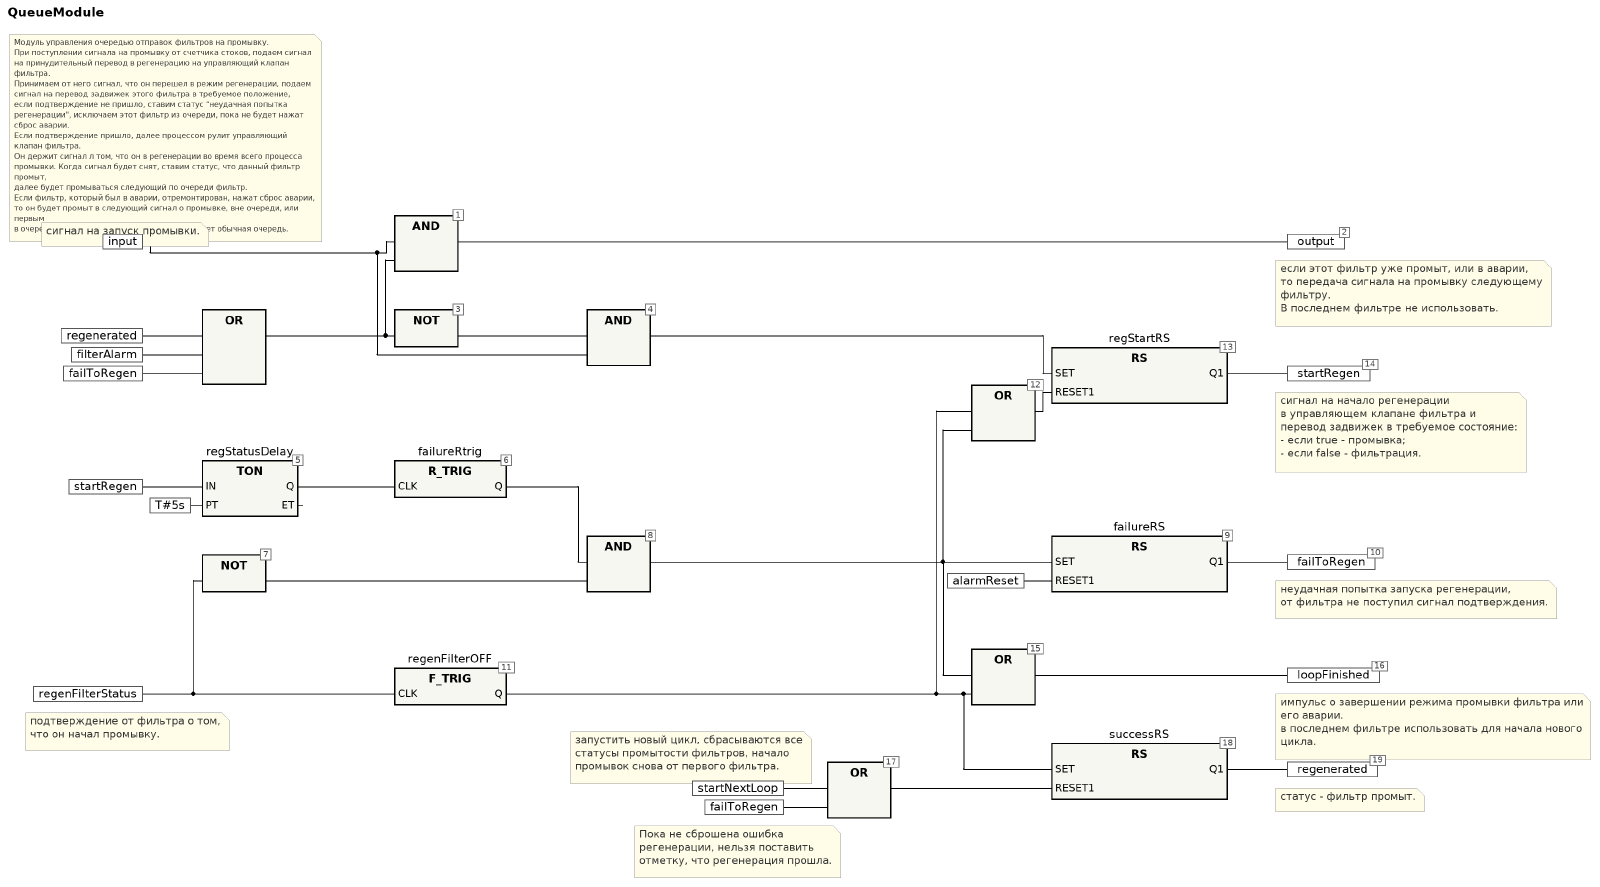
_CFC_ (* Continuous Function Chart, elements in execution order *)
(* Пока не сброшена ошибка / регенерации, нельзя поставить / отметку, что регенерация прошла. *)
(* запустить новый цикл, сбрасываются все / статусы промытости фильтров, начало / промывок снова от первого фильтра. *)
(* Модуль управления очередью отправок фильтров на промывку. / При поступлении сигнала на промывку от счетчика стоков, подаем сигнал на принудительный перевод в регенерацию на управляющий клапан фильтра. / Принимаем от него сигнал, что он перешел в режим регенерации, подаем сигнал на перевод задвижек этого фильтра в требуемое положение, / если подтверждение не пришло, ставим статус "неудачная попытка регенерации", исключаем этот фильтр из очереди, пока не будет нажат сброс аварии. / Если подтверждение пришло, далее процессом рулит управляющий клапан фильтра. / Он держит сигнал л том, что он в регенерации во время всего процесса промывки. Когда сигнал будет снят, ставим статус, что данный фильтр промыт, / далее будет промываться следующий по очереди фильтр. / Если фильтр, который был в аварии, отремонтирован, нажат сброс аварии, то он будет промыт в следующий сигнал о промывке, вне очереди, или первым / в очереди отремонтированных, после чего пойдет обычная очередь. *)
(* сигнал на запуск промывки. *)
(* если этот фильтр уже промыт, или в аварии, / то передача сигнала на промывку следующему фильтру. / В последнем фильтре не использовать. *)
(* сигнал на начало регенерации / в управляющем клапане фильтра и / перевод задвижек в требуемое состояние: / - если true - промывка; / - если false - фильтрация. *)
(* неудачная попытка запуска регенерации, / от фильтра не поступил сигнал подтверждения. *)
(* статус - фильтр промыт. *)
(* подтверждение от фильтра о том, / что он начал промывку. *)
(* импульс о завершении режима промывки фильтра или его аварии. / в последнем фильтре использовать для начала нового цикла. *)
#0 OR(regenerated, filterAlarm, failToRegen)
#1 AND(input, #0)
#2 output <= #1
#3 NOT(#0)
#4 AND(#3, input)
#5 regStatusDelay:TON(IN: startRegen, PT: T#5s)
#6 failureRtrig:R_TRIG(CLK: #5.Q)
#7 NOT(regenFilterStatus)
#8 AND(#6.Q, #7)
#9 failureRS:RS(SET: #8, RESET1: alarmReset)
#10 failToRegen <= #9.Q1
#11 regenFilterOFF:F_TRIG(CLK: regenFilterStatus)
#12 OR(#11.Q, #8)
#13 regStartRS:RS(SET: #4, RESET1: #12)
#14 startRegen <= #13.Q1
#15 OR(#8, #11.Q)
#16 loopFinished <= #15
#17 OR(startNextLoop, failToRegen)
#18 successRS:RS(SET: #11.Q, RESET1: #17)
#19 regenerated <= #18.Q1
_END_CFC_
(* the same logic as Structured Text *)
(* Пока не сброшена ошибка / регенерации, нельзя поставить / отметку, что регенерация прошла. *)
(* запустить новый цикл, сбрасываются все / статусы промытости фильтров, начало / промывок снова от первого фильтра. *)
(* Модуль управления очередью отправок фильтров на промывку. / При поступлении сигнала на промывку от счетчика стоков, подаем сигнал на принудительный перевод в регенерацию на управляющий клапан фильтра. / Принимаем от него сигнал, что он перешел в режим регенерации, подаем сигнал на перевод задвижек этого фильтра в требуемое положение, / если подтверждение не пришло, ставим статус "неудачная попытка регенерации", исключаем этот фильтр из очереди, пока не будет нажат сброс аварии. / Если подтверждение пришло, далее процессом рулит управляющий клапан фильтра. / Он держит сигнал л том, что он в регенерации во время всего процесса промывки. Когда сигнал будет снят, ставим статус, что данный фильтр промыт, / далее будет промываться следующий по очереди фильтр. / Если фильтр, который был в аварии, отремонтирован, нажат сброс аварии, то он будет промыт в следующий сигнал о промывке, вне очереди, или первым / в очереди отремонтированных, после чего пойдет обычная очередь. *)
(* сигнал на запуск промывки. *)
(* если этот фильтр уже промыт, или в аварии, / то передача сигнала на промывку следующему фильтру. / В последнем фильтре не использовать. *)
(* сигнал на начало регенерации / в управляющем клапане фильтра и / перевод задвижек в требуемое состояние: / - если true - промывка; / - если false - фильтрация. *)
(* неудачная попытка запуска регенерации, / от фильтра не поступил сигнал подтверждения. *)
(* статус - фильтр промыт. *)
(* подтверждение от фильтра о том, / что он начал промывку. *)
(* импульс о завершении режима промывки фильтра или его аварии. / в последнем фильтре использовать для начала нового цикла. *)
_t45 := regenerated OR filterAlarm OR failToRegen;
output := input AND _t45;
regStatusDelay(IN := startRegen, PT := T#5s);
failureRtrig(CLK := regStatusDelay.Q);
_t78 := failureRtrig.Q AND NOT regenFilterStatus;
failureRS(SET := _t78, RESET1 := alarmReset);
failToRegen := failureRS.Q1;
regenFilterOFF(CLK := regenFilterStatus);
regStartRS(SET := NOT _t45 AND input, RESET1 := regenFilterOFF.Q OR _t78);
startRegen := regStartRS.Q1;
loopFinished := _t78 OR regenFilterOFF.Q;
successRS(SET := regenFilterOFF.Q, RESET1 := startNextLoop OR failToRegen);
regenerated := successRS.Q1;
END_FUNCTION_BLOCK

(* POU SimpleValve, CFC *)
FUNCTION_BLOCK SimpleValve
VAR_INPUT
	inputOpen: BOOL;			(*вход для подачи импульса на открытие*)
	inputClose: BOOL;		(*вход для подачи импульса на закрытие*)
	statusOpen: BOOL;		(*статус: заслонка/задвижка ОТКРЫТА*)
	statusClose: BOOL;		(*статус: заслонка/задвижка ЗАКРЫТА*)
	reset: BOOL;		(*ручной сброс выходов и аварий в неактивное состояние*)
	timeToOpenClose: WORD;		(*Время в секундах на открытие/закрытие (по тех.характеристикам прибора).*)
END_VAR
VAR_OUTPUT
	outputOpen: BOOL;		(*выход на открытие задвижки/заслонки*)
	outputClose: BOOL;		(*выход на закрытие задвижки/заслонки*)
	errorToOpen: BOOL;		(*авария на открытие - задвижка не открылась за заданное время.*)
	errorToClose: BOOL;		(*авария на закрытие - задвижка не закрылась за заданное время.*)
END_VAR
VAR
	toOpenTrigger: RS;			(*Триггер сигнала на открытие.*)
	toCloseTrigger: RS;			(*Триггер сигнала на закрытие.*)
	timerToOpenClose: TON;		(*Таймер контроля времени открытия/закрытия.*)
	timerToStopOpening: TOF;		(*Задержка на останов открытия заслонки после получения статуса
										открыт от концевиков для плотного закрытия, полного открытия.*)
	timerToStopClosing: TOF;		(*Задержка на останов закрытия заслонки после получения статуса
										закрыт от концевиков для плотного закрытия, полного открытия.*)
	timerToDelayOpen: TOF;		(*Делает паузу 2,5 секунды на открытие после закрытия.*)
	timerToDelayClose: TOF;		(*Делает паузу 2,5 секунды на закрытие после открытия.*)
	statusOpenRS: RS;		(*Защелка сигнала об открытии*)
	statusCloseRS: RS;		(*Защелка сигнала о закрытии*)
END_VAR
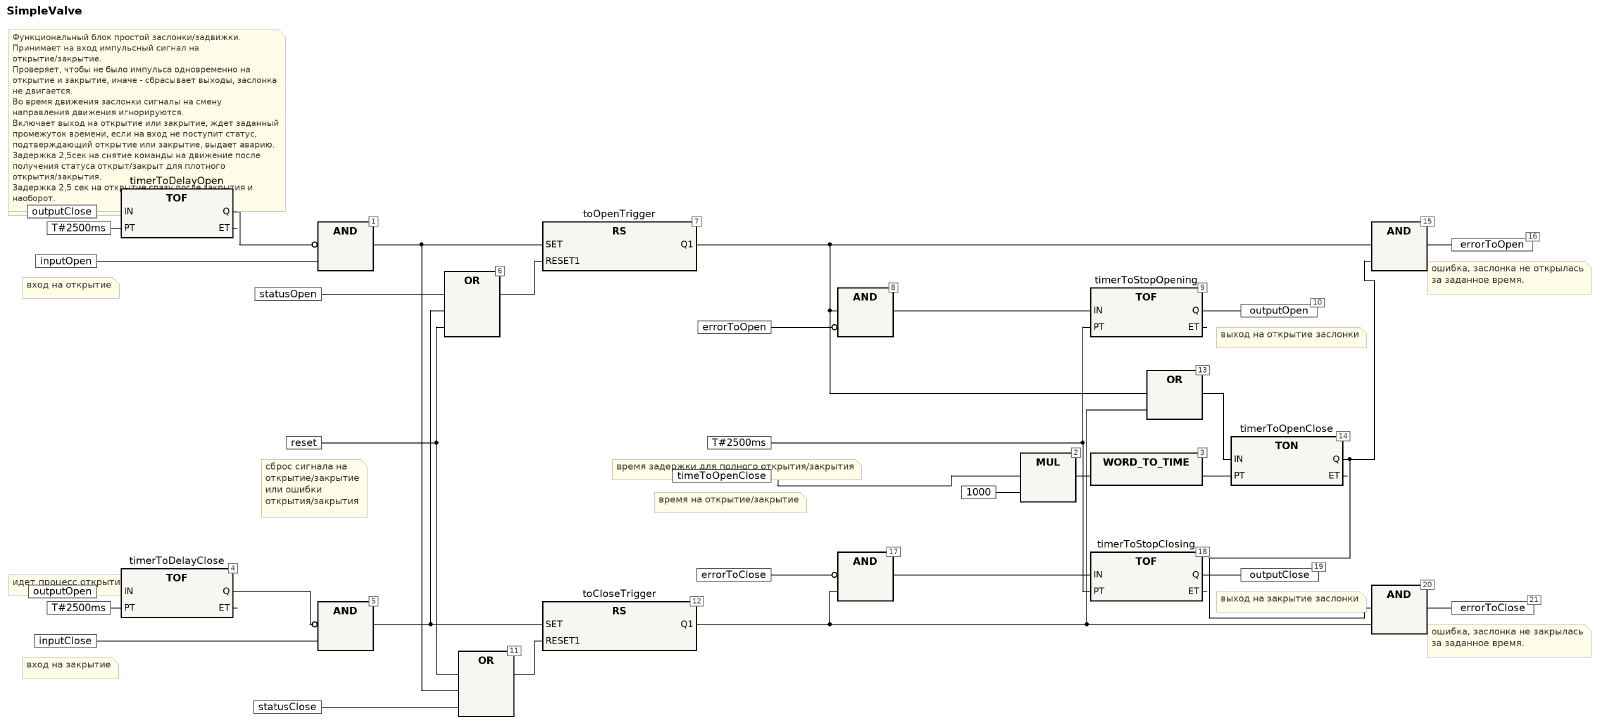
_CFC_ (* Continuous Function Chart, elements in execution order *)
(* идет процесс открытия *)
(* вход на закрытие *)
(* идет процесс закрытия *)
(* сброс сигнала на / открытие/закрытие / или ошибки / открытия/закрытия *)
(* вход на открытие *)
(* Функциональный блок простой заслонки/задвижки. / Принимает на вход импульсный сигнал на открытие/закрытие. / Проверяет, чтобы не было импульса одновременно на открытие и закрытие, иначе - сбрасывает выходы, заслонка не двигается. / Во время движения заслонки сигналы на смену направления движения игнорируются. / Включает выход на открытие или закрытие, ждет заданный промежуток времени, если на вход не поступит статус, подтверждающий открытие или закрытие, выдает аварию. / Задержка 2,5сек на снятие команды на движение после получения статуса открыт/закрыт для плотного открытия/закрытия. / Задержка 2,5 сек на открытие сразу после закрытия и наоборот. *)
(* время задержки для полного открытия/закрытия *)
(* время на открытие/закрытие *)
(* выход на открытие заслонки *)
(* ошибка, заслонка не открылась / за заданное время. *)
(* выход на закрытие заслонки *)
(* ошибка, заслонка не закрылась / за заданное время. *)
#0 timerToDelayOpen:TOF(IN: outputClose, PT: T#2500ms)
#1 AND(NOT #0.Q, inputOpen)
#2 MUL(timeToOpenClose, 1000)
#3 WORD_TO_TIME(#2)
#4 timerToDelayClose:TOF(IN: outputOpen, PT: T#2500ms)
#5 AND(NOT #4.Q, inputClose)
#6 OR(statusOpen, #5, reset)
#7 toOpenTrigger:RS(SET: #1, RESET1: #6)
#8 AND(#7.Q1, NOT errorToOpen)
#9 timerToStopOpening:TOF(IN: #8, PT: T#2500ms)
#10 outputOpen <= #9.Q
#11 OR(reset, #1, statusClose)
#12 toCloseTrigger:RS(SET: #5, RESET1: #11)
#13 OR(#7.Q1, #12.Q1)
#14 timerToOpenClose:TON(IN: #13, PT: #3)
#15 AND(#7.Q1, #14.Q)
#16 errorToOpen <= #15
#17 AND(NOT errorToClose, #12.Q1)
#18 timerToStopClosing:TOF(IN: #17, PT: T#2500ms)
#19 outputClose <= #18.Q
#20 AND(#14.Q, #12.Q1)
#21 errorToClose <= #20
_END_CFC_
END_FUNCTION_BLOCK

(* POU RichTwoPumpManager, CFC *)
FUNCTION_BLOCK RichTwoPumpManager
VAR_INPUT
	start: BOOL;		(*Сигнал на запуск насоса согласно выбранному режиму.*)
	setPump1main: BOOL;		(*Установить режим - насос 1 = главный.
Включать импульсом.*)
	setPump2main: BOOL;		(*Установить режим - насос 2 = главный.
Включать импульсом.*)
	setByCounter: BOOL;		(*Установить режим - по количеству включений.
Включать импульсом.*)
	setByWorkTime: BOOL;		(*Установить режим - по наработке.
Включать импульсом.*)
	resetPump1counter: BOOL;		(*Сброс счетчика количества включений насоса 1.*)
	resetPump2counter: BOOL;		(*Сброс счетчика количества включений насоса 2.*)
	resetWorkTimePump1: BOOL;		(*Сброс счетчика наработки насоса 1.*)
	resetWorkTimePump2: BOOL;		(*Сброс счетчика наработки насоса 2.*)
	startPump1man: BOOL;		(*Пуск насоса 1 вручную независимо от текущего режима.*)
	startPump2man: BOOL;		(*Пуск насоса 2 вручную независимо от текущего режима.*)
	stop: BOOL;		(*Стоп обоих насосов пока вход активен.
Не стоит применять для штатного останова.*)
	resetAlarms: BOOL;		(*Сброс аварий насоса.*)
	delayRepeatedStartTime: WORD;		(*Количество секунд на задержку повторного пуска насоса.
Защита от частых включений. Если ничего не подключено = 300сек.*)
	alarmPump1input: BOOL;		(*Вход от источника сигнала об аварии насоса 1.*)
	alarmPump2input: BOOL;		(*Вход от источника сигнала об аварии насоса 2.*)
END_VAR
VAR_OUTPUT
	regimePump1Main: BOOL;		(*Текущий режим - насос 1 = главный.*)
	regimePump2Main: BOOL;		(*Текущий режим - насос 2 = главный.*)
	regimeByCounter: BOOL;		(*Текущий режим - по количеству включений.*)
	regimeByWorkTime: BOOL;		(*Текущий режим - по наработке.*)
	counterPump1: DWORD;		(*Количество включений насоса 1.*)
	counterPump2: DWORD;		(*Количество включений насоса 2.*)
	daysPump1: WORD;		(*Количество отработанных дней насоса 1.*)
	hoursPump1: WORD;		(*Количество отработанных часов насоса 1.*)
	minutesPump1: WORD;		(*Количество отработанных минут насоса 1.*)
	secondsPump1: WORD;		(*Количество отработанных секунд насоса 1.*)
	daysPump2: WORD;		(*Количество отработанных дней насоса 2.*)
	hoursPump2: WORD;		(*Количество отработанных часов насоса 2.*)
	minutesPump2: WORD;		(*Количество отработанных минут насоса 2.*)
	secondsPump2: WORD;		(*Количество отработанных секунд насоса 2.*)
	pump1starter: BOOL;		(*Сигнал на запуск насоса 1.*)
	pump2starter: BOOL;		(*Сигнал на запуск насоса 2.*)
	nextStartP1timer: WORD;		(*Обратный отсчет до возможности повторного пуска насоса 1.*)
	nextStartP2timer: WORD;		(*Обратный отсчет до возможности повторного пуска насоса 2.*)
	alarmPump1output: BOOL;		(*Сигнал авария насоса 1.
Триггерится, нужен сброс.*)
	alarmPump2output: BOOL;		(*Сигнал авария насоса 2.
Триггерится, нужен сброс.*)
END_VAR
VAR
	ChoosePumpRegime: ChoosePumpRegime;		(*Блок выбора режима включения.*)
	CounterManager: CounterManager;		(*Блок выбора и запуска насоса по наработке.*)
	WorkTimeManager: WorkTimeManager;		(*Блок выбора и запуска насоса с меньшей наработкой.*)
	simpleTimeManager: SimpleTwoPumpManager;		(*Блок управления двумя насосами, горячий резерв, автоматическое переключение.*)
END_VAR
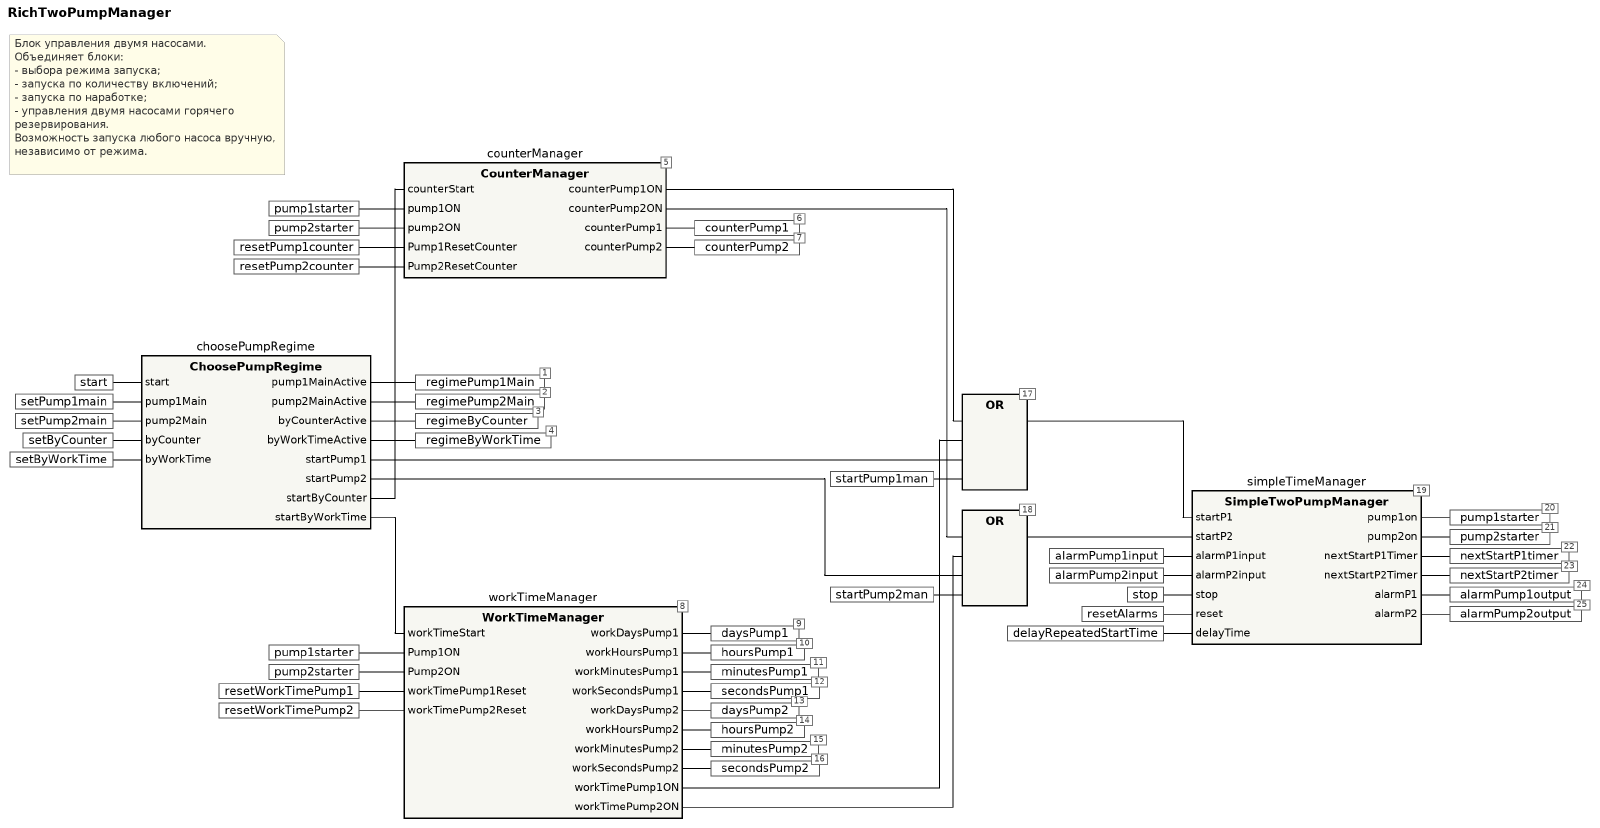
_CFC_ (* Continuous Function Chart, elements in execution order *)
(* Блок управления двумя насосами. / Объединяет блоки: / - выбора режима запуска; / - запуска по количеству включений; / - запуска по наработке; / - управления двумя насосами горячего резервирования. / Возможность запуска любого насоса вручную, / независимо от режима. *)
#0 choosePumpRegime:ChoosePumpRegime(start: start, pump1Main: setPump1main, pump2Main: setPump2main, byCounter: setByCounter, byWorkTime: setByWorkTime)
#1 regimePump1Main <= #0.pump1MainActive
#2 regimePump2Main <= #0.pump2MainActive
#3 regimeByCounter <= #0.byCounterActive
#4 regimeByWorkTime <= #0.byWorkTimeActive
#5 counterManager:CounterManager(counterStart: #0.startByCounter, pump1ON: pump1starter, pump2ON: pump2starter, Pump1ResetCounter: resetPump1counter, Pump2ResetCounter: resetPump2counter)
#6 counterPump1 <= #5.counterPump1
#7 counterPump2 <= #5.counterPump2
#8 workTimeManager:WorkTimeManager(workTimeStart: #0.startByWorkTime, Pump1ON: pump1starter, Pump2ON: pump2starter, workTimePump1Reset: resetWorkTimePump1, workTimePump2Reset: resetWorkTimePump2)
#9 daysPump1 <= #8.workDaysPump1
#10 hoursPump1 <= #8.workHoursPump1
#11 minutesPump1 <= #8.workMinutesPump1
#12 secondsPump1 <= #8.workSecondsPump1
#13 daysPump2 <= #8.workDaysPump2
#14 hoursPump2 <= #8.workHoursPump2
#15 minutesPump2 <= #8.workMinutesPump2
#16 secondsPump2 <= #8.workSecondsPump2
#17 OR(#5.counterPump1ON, #8.workTimePump1ON, #0.startPump1, startPump1man)
#18 OR(#5.counterPump2ON, #8.workTimePump2ON, #0.startPump2, startPump2man)
#19 simpleTimeManager:SimpleTwoPumpManager(startP1: #17, startP2: #18, alarmP1input: alarmPump1input, alarmP2input: alarmPump2input, stop: stop, reset: resetAlarms, delayTime: delayRepeatedStartTime)
#20 pump1starter <= #19.pump1on
#21 pump2starter <= #19.pump2on
#22 nextStartP1timer <= #19.nextStartP1Timer
#23 nextStartP2timer <= #19.nextStartP2Timer
#24 alarmPump1output <= #19.alarmP1
#25 alarmPump2output <= #19.alarmP2
_END_CFC_
(* the same logic as Structured Text *)
(* Блок управления двумя насосами. / Объединяет блоки: / - выбора режима запуска; / - запуска по количеству включений; / - запуска по наработке; / - управления двумя насосами горячего резервирования. / Возможность запуска любого насоса вручную, / независимо от режима. *)
choosePumpRegime(start := start, pump1Main := setPump1main, pump2Main := setPump2main, byCounter := setByCounter, byWorkTime := setByWorkTime);
regimePump1Main := choosePumpRegime.pump1MainActive;
regimePump2Main := choosePumpRegime.pump2MainActive;
regimeByCounter := choosePumpRegime.byCounterActive;
regimeByWorkTime := choosePumpRegime.byWorkTimeActive;
counterManager(counterStart := choosePumpRegime.startByCounter, pump1ON := pump1starter, pump2ON := pump2starter, Pump1ResetCounter := resetPump1counter, Pump2ResetCounter := resetPump2counter);
counterPump1 := counterManager.counterPump1;
counterPump2 := counterManager.counterPump2;
workTimeManager(workTimeStart := choosePumpRegime.startByWorkTime, Pump1ON := pump1starter, Pump2ON := pump2starter, workTimePump1Reset := resetWorkTimePump1, workTimePump2Reset := resetWorkTimePump2);
daysPump1 := workTimeManager.workDaysPump1;
hoursPump1 := workTimeManager.workHoursPump1;
minutesPump1 := workTimeManager.workMinutesPump1;
secondsPump1 := workTimeManager.workSecondsPump1;
daysPump2 := workTimeManager.workDaysPump2;
hoursPump2 := workTimeManager.workHoursPump2;
minutesPump2 := workTimeManager.workMinutesPump2;
secondsPump2 := workTimeManager.workSecondsPump2;
simpleTimeManager(startP1 := counterManager.counterPump1ON OR workTimeManager.workTimePump1ON OR choosePumpRegime.startPump1 OR startPump1man, startP2 := counterManager.counterPump2ON OR workTimeManager.workTimePump2ON OR choosePumpRegime.startPump2 OR startPump2man, alarmP1input := alarmPump1input, alarmP2input := alarmPump2input, stop := stop, reset := resetAlarms, delayTime := delayRepeatedStartTime);
pump1starter := simpleTimeManager.pump1on;
pump2starter := simpleTimeManager.pump2on;
nextStartP1timer := simpleTimeManager.nextStartP1Timer;
nextStartP2timer := simpleTimeManager.nextStartP2Timer;
alarmPump1output := simpleTimeManager.alarmP1;
alarmPump2output := simpleTimeManager.alarmP2;
END_FUNCTION_BLOCK

(* POU WorkTimeManager, CFC *)
FUNCTION_BLOCK WorkTimeManager
VAR
	workTimePump1: TimeSeparator;		(*Блок вывода времени наработки  насоса 1.*)
	workTimePump2: TimeSeparator;		(*Блок вывода времени наработки насоса 2.*)
	currentWorkTimePump1: DWORD;		(*Текущая наработка в секундах насоса 1.*)
	currentWorkTimePump2: DWORD;		(*Текущая наработка в секундах насоса 2.*)
	pulsarP1: PulsePerSec;		(*Генератор импульса в секунду для наработки насоса 1.*)
	pulsarP2: PulsePerSec;		(*Генератор импульса в секунду для наработки насоса 2.*)
	timeStartRtrig: R_TRIG;		(*Детектор переднего фронта сигнала на запуск.*)
	timeStartFtrig: F_TRIG;		(*Детектор спада сигнала на запуск.*)
	RStrigTimePump1: RS;		(*RSтриггер сигнала на запуск насоса 1.*)
	RStrigTimePump2: RS;		(*RSтриггер сигнала на запуск насоса 2.*)
END_VAR
VAR_OUTPUT
	workDaysPump1: WORD;		(*Количество отработанных дней для насоса 1.*)
	workHoursPump1: WORD;		(*Количество отработанных часов для насоса 1.*)
	workMinutesPump1: WORD;		(*Количество отработанных минут для насоса 1.*)
	workSecondsPump1: WORD;		(*Количество отработанных секунд для насоса 1.*)
	workDaysPump2: WORD;		(*Количество отработанных дней для насоса 2.*)
	workHoursPump2: WORD;		(*Количество отработанных часов для насоса 2.*)
	workMinutesPump2: WORD;		(*Количество отработанных минут для насоса 2.*)
	workSecondsPump2: WORD;		(*Количество отработанных секунд для насоса 2.*)
	workTimePump1ON: BOOL;		(*Выход на запуск насоса 1.*)
	workTimePump2ON: BOOL;		(*Выход на запуск насоса 2.*)
END_VAR
VAR_INPUT
	workTimeStart: BOOL;		(*Сигнал на запуск насоса с наименьшим временем работы.*)
	Pump1ON: BOOL;		(*Сигнал подтверждение о запуске насоса 1.*)
	Pump2ON: BOOL;		(*Сигнал подтверждение о запуске насоса 2.*)
	workTimePump1Reset: BOOL;		(*Сброс времени наработки насоса 1.*)
	workTimePump2Reset: BOOL;		(*Сброс времени наработки насоса 2.*)
END_VAR
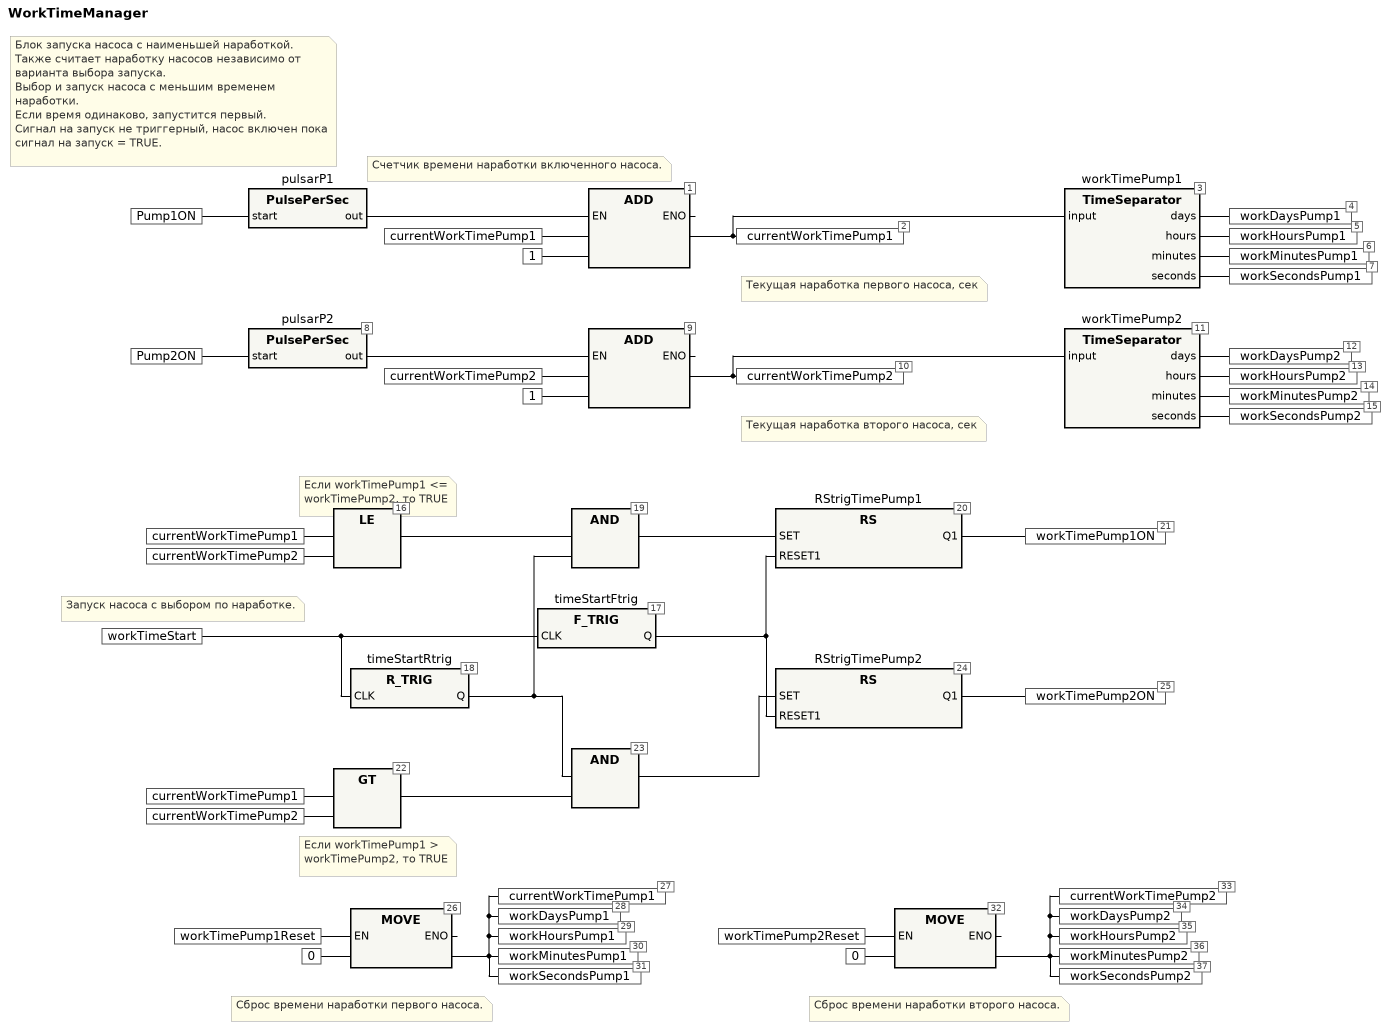
_CFC_ (* Continuous Function Chart, elements in execution order *)
(* Текущая наработка второго насоса, сек *)
(* Сброс времени наработки второго насоса. *)
(* Текущая наработка первого насоса, сек *)
(* Счетчик времени наработки включенного насоса. *)
(* Если workTimePump1 > / workTimePump2, то TRUE *)
(* Если workTimePump1 <= / workTimePump2, то TRUE *)
(* Запуск насоса с выбором по наработке. *)
(* Блок запуска насоса с наименьшей наработкой. / Также считает наработку насосов независимо от варианта выбора запуска. / Выбор и запуск насоса с меньшим временем наработки. / Если время одинаково, запустится первый. / Сигнал на запуск не триггерный, насос включен пока сигнал на запуск = TRUE. *)
(* Сброс времени наработки первого насоса. *)
#0 pulsarP1:PulsePerSec(start: Pump1ON)
#1 ADD(EN: #0.out, currentWorkTimePump1, 1)
#2 currentWorkTimePump1 <= #1
#3 workTimePump1:TimeSeparator(input: #1)
#4 workDaysPump1 <= #3.days
#5 workHoursPump1 <= #3.hours
#6 workMinutesPump1 <= #3.minutes
#7 workSecondsPump1 <= #3.seconds
#8 pulsarP2:PulsePerSec(start: Pump2ON)
#9 ADD(EN: #8.out, currentWorkTimePump2, 1)
#10 currentWorkTimePump2 <= #9
#11 workTimePump2:TimeSeparator(input: #9)
#12 workDaysPump2 <= #11.days
#13 workHoursPump2 <= #11.hours
#14 workMinutesPump2 <= #11.minutes
#15 workSecondsPump2 <= #11.seconds
#16 LE(currentWorkTimePump1, currentWorkTimePump2)
#17 timeStartFtrig:F_TRIG(CLK: workTimeStart)
#18 timeStartRtrig:R_TRIG(CLK: workTimeStart)
#19 AND(#16, #18.Q)
#20 RStrigTimePump1:RS(SET: #19, RESET1: #17.Q)
#21 workTimePump1ON <= #20.Q1
#22 GT(currentWorkTimePump1, currentWorkTimePump2)
#23 AND(#18.Q, #22)
#24 RStrigTimePump2:RS(SET: #23, RESET1: #17.Q)
#25 workTimePump2ON <= #24.Q1
#26 MOVE(EN: workTimePump1Reset, 0)
#27 currentWorkTimePump1 <= #26
#28 workDaysPump1 <= #26
#29 workHoursPump1 <= #26
#30 workMinutesPump1 <= #26
#31 workSecondsPump1 <= #26
#32 MOVE(EN: workTimePump2Reset, 0)
#33 currentWorkTimePump2 <= #32
#34 workDaysPump2 <= #32
#35 workHoursPump2 <= #32
#36 workMinutesPump2 <= #32
#37 workSecondsPump2 <= #32
_END_CFC_
END_FUNCTION_BLOCK

(* POU TimeSeparator, ST *)
FUNCTION_BLOCK TimeSeparator
VAR_INPUT
	 input: DWORD; (*Вход счетчика  наработки и т.п., сек.*)
END_VAR
VAR_OUTPUT
	days: WORD; (*Выход наработка, дней*)
	hours: WORD; (*Выход наработка, часов*)
	minutes: WORD; (*Выход наработка, минут*)
	seconds: WORD; (*Выход наработка, секунд*)
END_VAR
VAR
	temp: DWORD;
END_VAR
days:= DWORD_TO_WORD (input / (60 * 60 * 24));
temp:= input MOD (60 * 60 * 24);
hours:= DWORD_TO_WORD (temp / (60 * 60));
temp:= temp MOD (60 * 60);
minutes:= DWORD_TO_WORD (temp / 60);
temp:= temp MOD 60;
seconds:= DWORD_TO_WORD (temp);
END_FUNCTION_BLOCK

(* POU SimpleTwoPumpManager, CFC *)
FUNCTION_BLOCK SimpleTwoPumpManager

